FUNCTION_BLOCK FB 120
VERSION : 0.1
VAR_INPUT
  IN_Cm_ON : BOOL ;	//1: Attiva il ciclo; 0: Reset del ciclo
  IN_HOLD : BOOL ;	//Blocca il ciclo nel passo successivo
  IN_STEP : BOOL ;
END_VAR
VAR_OUTPUT
  OUT_St_CicloInCorso : BOOL ;
  OUT_St_CicloTerminatoOK : BOOL ;
  OUT_St_CicloTerminatoKO : BOOL ;
  OUT_CicloStato : INT ;
  OUT_Page : INT ;
  OUT_Message : INT ;
END_VAR
VAR
  Stato : INT ;
  StatoSeguente : INT ;
  FrontePassoSingolo : BOOL ;
  Stat_CicloTermOk : BOOL ;
  Stat_CicloTermKO : BOOL ;
  Stat_CicloInCorso : BOOL ;
  Timer_Pennarello : SFB 4;
END_VAR
VAR_TEMP
  Pag_Active : ARRAY  [0 .. 100 ] OF BOOL ;
END_VAR
BEGIN
NETWORK
TITLE = FLOW CHART
NETWORK
TITLE = Update state
      A     #IN_Cm_ON;
      JC    M002;
      L     0;
      T     #Stato;
      T     #StatoSeguente;
M002: NOP   0;
//->Update State
      A     #IN_STEP;
      FP    #FrontePassoSingolo;
      ON    #IN_HOLD;	//se usassi UN l'Hold agirebbe anche su avanzamento a passo singolo 
      JCN   N100;
      L     #StatoSeguente;
      T     #Stato;
N100: NOP   0;
// determinazione bit di stato
      CALL  FC 17 (
           Valore                   := #Stato,
           States                   := P#DB120.DBX 8.0 BYTE 8);
NETWORK
TITLE = Detect page active from OP
// serve??????
//      CALL  "Conv_INT->BIT"
//       Valore:=DB325.DBW2
//       States:=#Pag_Active
NETWORK
TITLE = States particular
      L     #Stato;
      L     0;
      <>I;
//->Evita ritardi
      A     #IN_Cm_ON;
      =     #Stat_CicloInCorso;
      A     DB120.DBX 15.4;
      =     #Stat_CicloTermOk;
      A     DB120.DBX 37.7;
      =     #Stat_CicloTermKO;
NETWORK
TITLE = Diagnostic default
//    L     0
//    T     #Page
//    L     0
//    T     #Message 
//      L     6
//      T     #StatoSeguente
NETWORK
TITLE = State <0>: Ciclo off
      A     DB120.DBX 8.0;
      A     #IN_Cm_ON;
      JC    A000;
      L     DB120.DBW 2;
      T     #OUT_Page;
      L     1;	// Ciclo off
      T     #OUT_Message;
      JU    Z000;
A000: L     10;
      T     #StatoSeguente;
Z000: NOP   0;
NETWORK
TITLE = State <10>: Inserimento pezzi su attrezzo e start ciclo
      A     DB120.DBX 9.2;
      JCN   Z010;
      A     DB101.DBX 0.6;
      A     DB101.DBX 0.4;
      A     DB106.DBX 0.7;
      A     DB106.DBX 1.0;
      AN    DB106.DBX 1.1;
      A     DB106.DBX 1.2;
      AN    DB106.DBX 1.3;
      A     DB106.DBX 1.4;
      AN    DB106.DBX 1.5;
      A     DB105.DBX 0.6;
      JC    Y010;
// Messaggi
// Inserisci spacer correttamente
      AN    DB106.DBX 1.0;
      ON    DB106.DBX 1.2;
      ON    DB106.DBX 1.4;
      JC    A010;
// almeno uno Spacer inserito male
      A     DB106.DBX 1.1;
      O     DB106.DBX 1.3;
      O     DB106.DBX 1.3;
      JC    B010;
// Inserisci nozzle ring
      AN    DB106.DBX 0.7;
      JC    C010;
// Start ciclo per Bloccare il pezzo
      JU    D010;
A010: L     DB120.DBW 2;
      T     #OUT_Page;
      L     2;	// Inserisci spacer correttamente
      T     #OUT_Message;
      JU    Z010;
B010: L     DB120.DBW 2;
      T     #OUT_Page;
      L     3;	// almeno uno Spacer inserito male
      T     #OUT_Message;
      JU    Z010;
C010: L     DB120.DBW 2;
      T     #OUT_Page;
      L     4;	// Inserisci nozzle ring
      T     #OUT_Message;
      JU    Z010;
D010: L     DB120.DBW 2;
      T     #OUT_Page;
      L     5;	// Start ciclo per Bloccare il pezzo
      T     #OUT_Message;
      JU    Z010;
// Stati di destinazione
Y010: L     13;
      T     #StatoSeguente;
Z010: NOP   0;
NETWORK
TITLE = State <13>: Blocca Pezzo e sblocca index
      A     DB120.DBX 9.5;
      JCN   Z013;
      A     DB101.DBX 0.5;
      A     DB101.DBX 0.3;
      A(;
      A     DB105.DBX 11.3;
      O     DB105.DBX 11.7;
      );
      A     DB105.DBX 10.2;
      JC    Y013;
// Messaggi
// Blocco pezzo e sblocco cassetto in corso
      AN    DB101.DBX 0.5;
      ON    DB101.DBX 0.3;
      JC    A013;
// Porta cassetto in zona di lavorazione
      AN    DB105.DBX 10.2;
      JC    B013;
      JU    B013;
A013: L     DB120.DBW 2;
      T     #OUT_Page;
      L     6;	// Blocco pezzo e sblocco cassetto in corso
      T     #OUT_Message;
      JU    Z013;
B013: L     DB120.DBW 2;
      T     #OUT_Page;
      L     7;	// Porta cassetto in zona di lavorazione
      T     #OUT_Message;
      JU    Z013;
// Stati di destinazione
Y013: L     16;
      T     #StatoSeguente;
Z013: NOP   0;
NETWORK
TITLE = State <16>: Blocca cassetto e prenota ribaditrice
      A     DB120.DBX 10.0;
      JCN   Z016;
      A     DB101.DBX 0.5;
      A     DB101.DBX 0.4;
      A     DB105.DBX 10.2;
      A     DB105.DBX 11.0;
      JC    Y016;
// Messaggi
// Blocco cassetto in corso
      AN    DB101.DBX 0.5;
      ON    DB101.DBX 0.4;
      ON    DB105.DBX 10.2;
      JC    A016;
// Attesa prenotazione ribaditrice
      AN    DB105.DBX 11.0;
      JC    B016;
      JU    B016;
A016: L     DB120.DBW 2;
      T     #OUT_Page;
      L     8;	// Blocco cassetto in corso
      T     #OUT_Message;
      JU    Z016;
B016: L     DB120.DBW 2;
      T     #OUT_Page;
      L     9;	//  Attesa prenotazione ribaditrice
      T     #OUT_Message;
      JU    Z016;
// Stati di destinazione
Y016: L     20;
      T     #StatoSeguente;
Z016: NOP   0;
NETWORK
TITLE = State <20>: Vai a quota di ribaditura punto corrente
      A     DB120.DBX 10.4;
      JCN   Z020;
      A     DB105.DBX 11.1;
      A     DB105.DBX 11.5;
      JC    Y020;
// Messaggi
// Posizionamento assi
      L     DB120.DBW 2;
      T     #OUT_Page;
      L     14;	// Posizionamento assi
      T     #OUT_Message;
      JU    Z020;
// Stati di destinazione
Y020: L     25;
      T     #StatoSeguente;
Z020: NOP   0;
NETWORK
TITLE = State <25>: Esegui ribaditura punto corrente
      A     DB120.DBX 11.1;
      JCN   Z025;
      A     DB105.DBX 11.2;
      JC    Y025;
// Messaggi
// Ribaditura spacer in corso
      L     DB120.DBW 2;
      T     #OUT_Page;
      L     9;	// Ribaditura spacer in corso
      T     #OUT_Message;
      JU    Z025;
// Stati di destinazione
Y025: L     30;
      T     #StatoSeguente;
Z025: NOP   0;
NETWORK
TITLE = State <30>: Risali ribaditrice
      A     DB120.DBX 11.6;
      JCN   Z030;
      A     DB105.DBX 11.3;
      A(;
      L     DB105.DBW 20;
      L     DB110.DBW 80;
      <I;
      );
      JC    Y030;
      A     DB105.DBX 11.3;
      A(;
      L     DB105.DBW 20;
      L     DB110.DBW 80;
      >=I;
      );
      JC    X030;
// Messaggi
// Ribaditura spacer in corso
      L     DB120.DBW 2;
      T     #OUT_Page;
      L     9;	// Ribaditura spacer in corso
      T     #OUT_Message;
      JU    Z030;
// Stati di destinazione
Y030: L     20;
      T     #StatoSeguente;
      JU    Z030;
X030: L     35;
      T     #StatoSeguente;
Z030: NOP   0;
NETWORK
TITLE = State <35>: Sblocco index e cassetto fuori
      A     DB120.DBX 12.3;
      JCN   Z035;
      A     DB101.DBX 0.3;
      A     DB105.DBX 10.3;
      JC    Y035;
// Messaggi
// Sblocco index in corso
      AN    DB101.DBX 0.3;
      JC    A035;
// Porta cassetto in zona di carico
      JU    B035;
A035: L     DB120.DBW 2;
      T     #OUT_Page;
      L     10;	// Sblocco index in corso
      T     #OUT_Message;
      JU    Z035;
B035: L     DB120.DBW 2;
      T     #OUT_Page;
      L     11;	// Porta cassetto in zona di carico
      T     #OUT_Message;
      JU    Z035;
// Stati di destinazione
Y035: L     40;
      T     #StatoSeguente;
Z035: NOP   0;
NETWORK
TITLE = State <40>: Sblocco pezzo e fine lavorazione
      A     DB120.DBX 13.0;
      JCN   Z040;
      A     DB101.DBX 0.4;
      A     DB101.DBX 0.6;
      A     DB105.DBX 10.3;
      AN    DB106.DBX 0.7;
      AN    DB106.DBX 1.0;
      AN    DB106.DBX 1.2;
      AN    DB106.DBX 1.4;
      JC    Y040;
// Messaggi
// Blocco index e sblocco pezzo in corso
      AN    DB101.DBX 0.4;
      ON    DB101.DBX 0.6;
      JC    A040;
// Rimuovi pezzo buono dalla stazione
      JU    B040;
A040: L     DB120.DBW 2;
      T     #OUT_Page;
      L     12;	// Blocco index e sblocco pezzo in corso
      T     #OUT_Message;
      JU    Z040;
B040: L     DB120.DBW 2;
      T     #OUT_Page;
      L     13;	// Rimuovi pezzo buono dalla stazione
      T     #OUT_Message;
      JU    Z040;
// Stati di destinazione
Y040: L     60;
      T     #StatoSeguente;
Z040: NOP   0;
NETWORK
TITLE =
      A     DB120.DBX 15.4;
      JCN   Z060;
// Stati di destinazione
      L     10;
      T     #StatoSeguente;
Z060: NOP   0;
NETWORK
TITLE = Output
      L     #Stato;
      T     #OUT_CicloStato;
      A     #Stat_CicloInCorso;
      =     #OUT_St_CicloInCorso;
      A     #Stat_CicloTermOk;
      =     #OUT_St_CicloTerminatoOK;
      A     #Stat_CicloTermKO;
      =     #OUT_St_CicloTerminatoKO;
END_FUNCTION_BLOCK

FUNCTION_BLOCK FB 121
VERSION : 0.1
VAR_INPUT
  IN_Cm_ON : BOOL ;	//1: Attiva il ciclo; 0: Reset del ciclo
  IN_HOLD : BOOL ;	//Blocca il ciclo nel passo successivo
  IN_STEP : BOOL ;
END_VAR
VAR_OUTPUT
  OUT_St_CicloInCorso : BOOL ;
  OUT_St_CicloTerminatoOK : BOOL ;
  OUT_St_CicloTerminatoKO : BOOL ;
  OUT_CicloStato : INT ;
  OUT_Page : INT ;
  OUT_Message : INT ;
END_VAR
VAR
  Stato : INT ;
  StatoSeguente : INT ;
  FrontePassoSingolo : BOOL ;
  Stat_CicloTermOk : BOOL ;
  Stat_CicloTermKO : BOOL ;
  Stat_CicloInCorso : BOOL ;
  Timer_Pennarello : SFB 4;
END_VAR
VAR_TEMP
  Pag_Active : ARRAY  [0 .. 100 ] OF BOOL ;
END_VAR
BEGIN
NETWORK
TITLE = FLOW CHART
NETWORK
TITLE = Update state
      A     #IN_Cm_ON;
      JC    M002;
      L     0;
      T     #Stato;
      T     #StatoSeguente;
M002: NOP   0;
//->Update State
      A     #IN_STEP;
      FP    #FrontePassoSingolo;
      ON    #IN_HOLD;	//se usassi UN l'Hold agirebbe anche su avanzamento a passo singolo 
      JCN   N100;
      L     #StatoSeguente;
      T     #Stato;
N100: NOP   0;
// determinazione bit di stato
      CALL  FC 17 (
           Valore                   := #Stato,
           States                   := P#DB120.DBX 30.0 BYTE 8);
NETWORK
TITLE = States particular
      L     #Stato;
      L     0;
      <>I;
//->Evita ritardi
      A     #IN_Cm_ON;
      =     #Stat_CicloInCorso;
      A     DB120.DBX 37.4;
      =     #Stat_CicloTermOk;
      A     DB120.DBX 37.7;
      =     #Stat_CicloTermKO;
NETWORK
TITLE = State <0>: Ciclo off
      A     DB120.DBX 30.0;
      A     #IN_Cm_ON;
      JC    A000;
      L     DB120.DBW 24;
      T     #OUT_Page;
      L     20;	// ciclo off
      T     #OUT_Message;
      JU    Z000;
A000: L     10;
      T     #StatoSeguente;
Z000: NOP   0;
NETWORK
TITLE = State <10>: Sali ribaditrice
      A     DB120.DBX 31.2;
      JCN   Z010;
      A     DB105.DBX 11.3;
      O     DB105.DBX 11.7;
      AN    DB101.DBX 0.1;
      JC    Y010;
      A     DB105.DBX 11.3;
      O     DB105.DBX 11.7;
      A     DB101.DBX 0.1;
      JC    X010;
// Messaggi
// Salita ribaditrice in corso
      L     DB120.DBW 24;
      T     #OUT_Page;
      L     21;	// Salita ribaditrice in corso
      T     #OUT_Message;
      JU    Z010;
// Stati di destinazione
Y010: L     15;
      T     #StatoSeguente;
      JU    Z010;
X010: L     20;
      T     #StatoSeguente;
Z010: NOP   0;
NETWORK
TITLE = State <15>: Sblocca index e cassetto fuori
      A     DB120.DBX 31.7;
      JCN   Z015;
      A     DB101.DBX 0.3;
      A     DB105.DBX 10.3;
      JC    Y015;
// Messaggi
//   Sblocco index in corso
      AN    DB101.DBX 0.3;
      JC    A015;
// Porta cassetto in zona di scarico
      JU    B015;
A015: L     DB120.DBW 24;
      T     #OUT_Page;
      L     22;	//  Sblocco index in corso
      T     #OUT_Message;
      JU    Z015;
B015: L     DB120.DBW 24;
      T     #OUT_Page;
      L     23;	// Porta cassetto in zona di scarico
      T     #OUT_Message;
      JU    Z015;
// Stati di destinazione
Y015: L     20;
      T     #StatoSeguente;
Z015: NOP   0;
NETWORK
TITLE = State <20>: Blocca index e sblocca pezzo - rimuovi scarto
      A     DB120.DBX 32.4;
      JCN   Z020;
      A     DB101.DBX 0.6;
      A     DB101.DBX 0.4;
      A     DB105.DBX 10.3;
      AN    DB106.DBX 0.7;
      JC    Y020;
// Messaggi
// Blocco index e sblocco pezzo in corso
      AN    DB101.DBX 0.6;
      ON    DB101.DBX 0.4;
      ON    DB105.DBX 10.3;
      JC    A020;
// Rimuovi pezzo scarto dalla stazione
      JU    B020;
A020: L     DB120.DBW 24;
      T     #OUT_Page;
      L     24;	// Blocco index e sblocco pezzo in corso
      T     #OUT_Message;
      JU    Z020;
B020: L     DB120.DBW 24;
      T     #OUT_Page;
      L     25;	// Rimuovi pezzo scarto dalla stazione
      T     #OUT_Message;
      JU    Z020;
// Stati di destinazione
Y020: L     60;
      T     #StatoSeguente;
Z020: NOP   0;
NETWORK
TITLE = Output
      L     #Stato;
      T     #OUT_CicloStato;
      A     #Stat_CicloInCorso;
      =     #OUT_St_CicloInCorso;
      A     #Stat_CicloTermOk;
      =     #OUT_St_CicloTerminatoOK;
      A     #Stat_CicloTermKO;
      =     #OUT_St_CicloTerminatoKO;
END_FUNCTION_BLOCK

FUNCTION_BLOCK FB 170
VERSION : 0.1
VAR_INPUT
  IN_Cm_ON : BOOL ;	//1: Attiva il ciclo; 0: Reset del ciclo
  IN_HOLD : BOOL ;	//Blocca il ciclo nel passo successivo
  IN_STEP : BOOL ;
END_VAR
VAR_OUTPUT
  OUT_St_CicloInCorso : BOOL ;
  OUT_St_CicloTerminatoOK : BOOL ;
  OUT_St_CicloTerminatoKO : BOOL ;
  OUT_CicloStato : INT ;
  OUT_Page : INT ;
  OUT_Message : INT ;
END_VAR
VAR
  Stato : INT ;
  StatoSeguente : INT ;
  FrontePassoSingolo : BOOL ;
  Stat_CicloTermOk : BOOL ;
  Stat_CicloTermKO : BOOL ;
  Stat_CicloInCorso : BOOL ;
END_VAR
VAR_TEMP
  Pag_Active : ARRAY  [0 .. 100 ] OF BOOL ;
END_VAR
BEGIN
NETWORK
TITLE = FLOW CHART
NETWORK
TITLE = Update state
      A     #IN_Cm_ON;
      JC    M002;
      L     0;
      T     #Stato;
      T     #StatoSeguente;
M002: NOP   0;
//->Update State
      A     #IN_STEP;
      FP    #FrontePassoSingolo;
      ON    #IN_HOLD;	//se usassi UN l'Hold agirebbe anche su avanzamento a passo singolo 
      JCN   N100;
      L     #StatoSeguente;
      T     #Stato;
N100: NOP   0;
// determinazione bit di stato
      CALL  FC 17 (
           Valore                   := #Stato,
           States                   := P#DB170.DBX 8.0 BYTE 8);
NETWORK
TITLE = States particular
      L     #Stato;
      L     0;
      <>I;
//->Evita ritardi
      A     #IN_Cm_ON;
      =     #Stat_CicloInCorso;
      A     DB170.DBX 15.4;
      =     #Stat_CicloTermOk;
      A     DB170.DBX 37.7;
      =     #Stat_CicloTermKO;
NETWORK
TITLE = Diagnostic default
NETWORK
TITLE = State <0>: Ciclo off
      A     DB170.DBX 8.0;
      A     #IN_Cm_ON;
      JC    A000;
      L     DB170.DBW 2;
      T     #OUT_Page;
      L     1;	// Ciclo off
      T     #OUT_Message;
      JU    Z000;
A000: L     10;
      T     #StatoSeguente;
Z000: NOP   0;
NETWORK
TITLE = State <10>: Inserimento pezzi su attrezzo e cassetto dentrro
      A     DB151.DBX 0.2;
      FP    M 52.0;
      =     DB155.DBX 11.7;
      A     DB155.DBX 11.7;
      A     DB170.DBX 9.2;
      S     DB155.DBX 12.0;
      A     DB155.DBX 12.0;
      AN    DB151.DBX 0.2;
      ON    DB170.DBX 9.2;
      R     DB155.DBX 12.0;
      A     DB155.DBX 12.0;
      L     S5T#500MS;
      SD    T 20;
      A     DB170.DBX 9.2;
      JCN   Z010;
      A     T 20;
      JC    Y010;
// Messaggi
// Inserisci pezzi e porta cassetto dentro
      L     DB170.DBW 2;
      T     #OUT_Page;
      L     2;	//  Inserisci pezzi e porta cassetto dentro
      T     #OUT_Message;
      JU    Z010;
// Stati di destinazione
Y010: L     15;
      T     #StatoSeguente;
Z010: NOP   0;
NETWORK
TITLE = State <15>: Blocca cassetto dentrro
      A     DB170.DBX 9.7;
      JCN   Z015;
      A     DB151.DBX 0.2;
      A     DB151.DBX 0.4;
      JC    Y015;
// Messaggi
// Blocco cassetto in corso
      L     DB170.DBW 2;
      T     #OUT_Page;
      L     3;	// Blocco cassetto in corso
      T     #OUT_Message;
      JU    Z015;
// Stati di destinazione
Y015: L     20;
      T     #StatoSeguente;
Z015: NOP   0;
NETWORK
TITLE = State <20>: Discesa gruppo di piantaggio
      A     DB170.DBX 10.4;
      JCN   Z020;
      A     DB151.DBX 0.7;
      JC    Y020;
// Messaggi
// Discesa gruppo di piantaggio
      L     DB170.DBW 2;
      T     #OUT_Page;
      L     4;	// Discesa gruppo di piantaggio
      T     #OUT_Message;
      JU    Z020;
// Stati di destinazione
Y020: L     25;
      T     #StatoSeguente;
Z020: NOP   0;
NETWORK
TITLE = State <25>: Discesa piantaggio
      A     DB170.DBX 11.1;
      JCN   Z025;
      A     DB155.DBX 11.2;
      JC    Y025;
// Messaggi
// Piantaggio in corso
      L     DB170.DBW 2;
      T     #OUT_Page;
      L     5;	// Piantaggio in corso
      T     #OUT_Message;
      JU    Z025;
// Stati di destinazione
Y025: L     30;
      T     #StatoSeguente;
Z025: NOP   0;
NETWORK
TITLE = State <30>: Risalita piantaggio
      A     DB170.DBX 11.6;
      JCN   Z030;
      A     DB151.DBX 1.0;
      A     DB151.DBX 0.6;
      JC    Y030;
// Messaggi
// Risalita pressa in corso
      L     DB170.DBW 2;
      T     #OUT_Page;
      L     6;	// Risalita pressa in corso
      T     #OUT_Message;
      JU    Z030;
// Stati di destinazione
Y030: L     35;
      T     #StatoSeguente;
Z030: NOP   0;
NETWORK
TITLE = State <35>: Sblocco cassetto
      A     DB170.DBX 12.3;
      JCN   Z035;
      A     DB151.DBX 0.3;
      JC    Y035;
// Messaggi
// Sblocco cassetto in corso
      L     DB170.DBW 2;
      T     #OUT_Page;
      L     7;	// Sblocco cassetto in corso
      T     #OUT_Message;
      JU    Z035;
// Stati di destinazione
Y035: L     60;
      T     #StatoSeguente;
Z035: NOP   0;
NETWORK
TITLE =
      A     DB170.DBX 15.4;
      JCN   Z060;
      L     10;
      T     #StatoSeguente;
Z060: NOP   0;
NETWORK
TITLE = Output
      L     #Stato;
      T     #OUT_CicloStato;
      A     #Stat_CicloInCorso;
      =     #OUT_St_CicloInCorso;
      A     #Stat_CicloTermOk;
      =     #OUT_St_CicloTerminatoOK;
      A     #Stat_CicloTermKO;
      =     #OUT_St_CicloTerminatoKO;
END_FUNCTION_BLOCK

FUNCTION_BLOCK FB 171
VERSION : 0.1
VAR_INPUT
  IN_Cm_ON : BOOL ;	//1: Attiva il ciclo; 0: Reset del ciclo
  IN_HOLD : BOOL ;	//Blocca il ciclo nel passo successivo
  IN_STEP : BOOL ;
END_VAR
VAR_OUTPUT
  OUT_St_CicloInCorso : BOOL ;
  OUT_St_CicloTerminatoOK : BOOL ;
  OUT_St_CicloTerminatoKO : BOOL ;
  OUT_CicloStato : INT ;
  OUT_Page : INT ;
  OUT_Message : INT ;
END_VAR
VAR
  Stato : INT ;
  StatoSeguente : INT ;
  FrontePassoSingolo : BOOL ;
  Stat_CicloTermOk : BOOL ;
  Stat_CicloTermKO : BOOL ;
  Stat_CicloInCorso : BOOL ;
END_VAR
VAR_TEMP
  Pag_Active : ARRAY  [0 .. 100 ] OF BOOL ;
END_VAR
BEGIN
NETWORK
TITLE = FLOW CHART
NETWORK
TITLE = Update state
      A     #IN_Cm_ON;
      JC    M002;
      L     0;
      T     #Stato;
      T     #StatoSeguente;
M002: NOP   0;
//->Update State
      A     #IN_STEP;
      FP    #FrontePassoSingolo;
      ON    #IN_HOLD;	//se usassi UN l'Hold agirebbe anche su avanzamento a passo singolo 
      JCN   N100;
      L     #StatoSeguente;
      T     #Stato;
N100: NOP   0;
// determinazione bit di stato
      CALL  FC 17 (
           Valore                   := #Stato,
           States                   := P#DB170.DBX 30.0 BYTE 8);
NETWORK
TITLE = States particular
      L     #Stato;
      L     0;
      <>I;
//->Evita ritardi
      A     #IN_Cm_ON;
      =     #Stat_CicloInCorso;
      A     DB170.DBX 37.4;
      =     #Stat_CicloTermOk;
      A     DB170.DBX 37.7;
      =     #Stat_CicloTermKO;
NETWORK
TITLE = Diagnostic default
NETWORK
TITLE = State <0>: Ciclo off
      A     DB170.DBX 30.0;
      A     #IN_Cm_ON;
      JC    A000;
      L     DB170.DBW 24;
      T     #OUT_Page;
      L     1;	// Ciclo off
      T     #OUT_Message;
      JU    Z000;
A000: L     10;
      T     #StatoSeguente;
Z000: NOP   0;
NETWORK
TITLE = State <10>: Risalita piantaggio
      A     DB170.DBX 31.2;
      JCN   Z010;
      A     DB151.DBX 1.0;
      A     DB151.DBX 0.6;
      JC    Y010;
// Messaggi
// Risalita pressa in corso
      L     DB170.DBW 24;
      T     #OUT_Page;
      L     6;	// Risalita pressa in corso
      T     #OUT_Message;
      JU    Z010;
// Stati di destinazione
Y010: L     15;
      T     #StatoSeguente;
Z010: NOP   0;
NETWORK
TITLE = State <15>: Sblocco cassetto
      A     DB170.DBX 31.7;
      JCN   Z015;
      A     DB151.DBX 0.3;
      JC    Y015;
// Messaggi
// Sblocco cassetto in corso
      L     DB170.DBW 24;
      T     #OUT_Page;
      L     7;	// Sblocco cassetto in corso
      T     #OUT_Message;
      JU    Z015;
// Stati di destinazione
Y015: L     60;
      T     #StatoSeguente;
Z015: NOP   0;
NETWORK
TITLE = Output
      L     #Stato;
      T     #OUT_CicloStato;
      A     #Stat_CicloInCorso;
      =     #OUT_St_CicloInCorso;
      A     #Stat_CicloTermOk;
      =     #OUT_St_CicloTerminatoOK;
      A     #Stat_CicloTermKO;
      =     #OUT_St_CicloTerminatoKO;
END_FUNCTION_BLOCK

FUNCTION_BLOCK FB 220
VERSION : 0.1
VAR_INPUT
  IN_Cm_ON : BOOL ;	//1: Attiva il ciclo; 0: Reset del ciclo
  IN_HOLD : BOOL ;	//Blocca il ciclo nel passo successivo
  IN_STEP : BOOL ;
END_VAR
VAR_OUTPUT
  OUT_St_CicloInCorso : BOOL ;
  OUT_St_CicloTerminatoOK : BOOL ;
  OUT_St_CicloTerminatoKO : BOOL ;
  OUT_CicloStato : INT ;
  OUT_Page : INT ;
  OUT_Message : INT ;
END_VAR
VAR
  Stato : INT ;
  StatoSeguente : INT ;
  FrontePassoSingolo : BOOL ;
  Stat_CicloTermOk : BOOL ;
  Stat_CicloTermKO : BOOL ;
  Stat_CicloInCorso : BOOL ;
  Timer_Pennarello : SFB 4;
END_VAR
VAR_TEMP
  Pag_Active : ARRAY  [0 .. 100 ] OF BOOL ;
END_VAR
BEGIN
NETWORK
TITLE = FLOW CHART
NETWORK
TITLE = Update state
      A     #IN_Cm_ON;
      JC    M002;
      L     0;
      T     #Stato;
      T     #StatoSeguente;
M002: NOP   0;
//->Update State
      A     #IN_STEP;
      FP    #FrontePassoSingolo;
      ON    #IN_HOLD;	//se usassi UN l'Hold agirebbe anche su avanzamento a passo singolo 
      JCN   N100;
      L     #StatoSeguente;
      T     #Stato;
N100: NOP   0;
// determinazione bit di stato
      CALL  FC 17 (
           Valore                   := #Stato,
           States                   := P#DB220.DBX 8.0 BYTE 8);
NETWORK
TITLE = Detect page active from OP
// serve??????
//      CALL  "Conv_INT->BIT"
//       Valore:=DB325.DBW2
//       States:=#Pag_Active
NETWORK
TITLE = States particular
      L     #Stato;
      L     0;
      <>I;
//->Evita ritardi
      A     #IN_Cm_ON;
      =     #Stat_CicloInCorso;
      A     DB220.DBX 15.4;
      =     #Stat_CicloTermOk;
      A     DB220.DBX 15.7;
      =     #Stat_CicloTermKO;
NETWORK
TITLE = Diagnostic default
//    L     0
//    T     #Page
//    L     0
//    T     #Message 
//      L     6
//      T     #StatoSeguente
NETWORK
TITLE = State <0>: Ciclo off
      A     DB220.DBX 8.0;
      A     #IN_Cm_ON;
      JC    A000;
      L     DB120.DBW 24;
      T     #OUT_Page;
      L     1;	// ciclo off
      T     #OUT_Message;
      JU    Z000;
A000: L     10;
      T     #StatoSeguente;
Z000: NOP   0;
NETWORK
TITLE = State <10>: Inserimento pezzi su attrezzo e start ciclo
      A     DB220.DBX 9.2;
      JCN   Z010;
      A     DB201.DBX 0.7;
      A     DB201.DBX 0.5;
      A     DB205.DBX 0.6;
      JC    Y010;
// Messaggi
// Inserisci nozzle ring e Start ciclo
      L     DB220.DBW 2;
      T     #OUT_Page;
      L     4;	// Inserisci nozzle ring e start ciclo
      T     #OUT_Message;
      JU    Z010;
// Stati di destinazione
Y010: L     11;
      T     #StatoSeguente;
Z010: NOP   0;
NETWORK
TITLE = State <11>: Blocca index e controlla presenza pezzo
      A     DB220.DBX 9.3;
      JCN   Z011;
      A     DB201.DBX 0.6;
      A     DB206.DBX 0.7;
      JC    Y011;
      A     DB205.DBX 0.6;
      JC    X011;
// Messaggi
// Inserisci nozzle ring
      AN    DB206.DBX 0.7;
      JC    A011;
      JU    Z011;
A011: L     DB220.DBW 2;
      T     #OUT_Page;
      L     5;	// Inserisci nozzle ring
      T     #OUT_Message;
      JU    Z011;
// Stati di destinazione
X011: L     10;
      T     #StatoSeguente;
      JU    Z011;
Y011: L     13;
      T     #StatoSeguente;
Z011: NOP   0;
NETWORK
TITLE = State <13>: sblocca index
      A     DB220.DBX 9.5;
      JCN   Z013;
      A     DB201.DBX 0.6;
      A     DB201.DBX 0.4;
      A(;
      A     DB205.DBX 11.3;
      O     DB205.DBX 11.7;
      );
      A     DB205.DBX 10.2;
      A     DB201.DBX 0.1;
      JC    Y013;
// Messaggi
// Blocco pezzo e sblocco cassetto in corso
      AN    DB201.DBX 0.6;
      ON    DB201.DBX 0.4;
      JC    A013;
// Porta cassetto in zona di lavorazione
      AN    DB205.DBX 10.2;
      JC    B013;
      JU    C013;
A013: L     DB220.DBW 2;
      T     #OUT_Page;
      L     6;	// Blocco pezzo e sblocco cassetto in corso
      T     #OUT_Message;
      JU    Z013;
B013: L     DB220.DBW 2;
      T     #OUT_Page;
      L     7;	// Porta cassetto in zona di lavorazione
      T     #OUT_Message;
      JU    Z013;
C013: L     DB220.DBW 2;
      T     #OUT_Page;
      L     3;	// Controlla presenza Pipe
      T     #OUT_Message;
      JU    Z013;
// Stati di destinazione
Y013: L     16;
      T     #StatoSeguente;
Z013: NOP   0;
NETWORK
TITLE = State <16>: Blocca cassetto e prenota ribaditrice
      A     DB220.DBX 10.0;
      JCN   Z016;
      A     DB201.DBX 0.6;
      A     DB201.DBX 0.5;
      A     DB205.DBX 10.2;
      A     DB205.DBX 11.0;
      JC    Y016;
// Messaggi
// Blocco cassetto in corso
      AN    DB201.DBX 0.6;
      ON    DB201.DBX 0.5;
      ON    DB205.DBX 10.2;
      JC    A016;
// Attesa prenotazione ribaditrice
      AN    DB205.DBX 11.0;
      JC    B016;
      JU    B016;
A016: L     DB220.DBW 2;
      T     #OUT_Page;
      L     8;	// Blocco cassetto in corso
      T     #OUT_Message;
      JU    Z016;
B016: L     DB220.DBW 2;
      T     #OUT_Page;
      L     9;	//  Attesa prenotazione ribaditrice
      T     #OUT_Message;
      JU    Z016;
// Stati di destinazione
Y016: L     20;
      T     #StatoSeguente;
Z016: NOP   0;
NETWORK
TITLE = State <20>: Vai a quota di ribaditura punto corrente
      A     DB220.DBX 10.4;
      JCN   Z020;
      A     DB205.DBX 11.1;
      A     DB205.DBX 11.5;
      JC    Y020;
// Messaggi
// Posizionamento assi
      L     DB220.DBW 2;
      T     #OUT_Page;
      L     15;	// Posizionamento assi
      T     #OUT_Message;
      JU    Z020;
// Stati di destinazione
Y020: L     25;
      T     #StatoSeguente;
Z020: NOP   0;
NETWORK
TITLE = State <25>: Esegui ribaditura punto corrente
      A     DB220.DBX 11.1;
      JCN   Z025;
      A     DB205.DBX 11.2;
      JC    Y025;
// Messaggi
// Ribaditura spacer in corso
      L     DB220.DBW 2;
      T     #OUT_Page;
      L     10;	// Ribaditura spacer in corso
      T     #OUT_Message;
      JU    Z025;
// Stati di destinazione
Y025: L     30;
      T     #StatoSeguente;
Z025: NOP   0;
NETWORK
TITLE = State <30>: Risali ribaditrice
      A     DB220.DBX 11.6;
      JCN   Z030;
      A     DB205.DBX 11.3;
      A(;
      L     DB205.DBW 20;
      L     DB210.DBW 80;
      <I;
      );
      JC    Y030;
      A     DB205.DBX 11.3;
      A(;
      L     DB205.DBW 20;
      L     DB210.DBW 80;
      >=I;
      );
      JC    X030;
// Messaggi
// Ribaditura spacer in corso
      L     DB220.DBW 2;
      T     #OUT_Page;
      L     10;	// Ribaditura spacer in corso
      T     #OUT_Message;
      JU    Z030;
// Stati di destinazione
Y030: L     20;
      T     #StatoSeguente;
      JU    Z030;
X030: L     35;
      T     #StatoSeguente;
Z030: NOP   0;
NETWORK
TITLE = State <35>: Sblocco index e cassetto fuori
      A     DB220.DBX 12.3;
      JCN   Z035;
      A     DB201.DBX 0.4;
      A     DB205.DBX 10.3;
      JC    Y035;
// Messaggi
// Sblocco index in corso
      AN    DB201.DBX 0.4;
      JC    A035;
// Porta cassetto in zona di carico
      JU    B035;
A035: L     DB220.DBW 2;
      T     #OUT_Page;
      L     11;	// Sblocco index in corso
      T     #OUT_Message;
      JU    Z035;
B035: L     DB220.DBW 2;
      T     #OUT_Page;
      L     12;	// Porta cassetto in zona di carico
      T     #OUT_Message;
      JU    Z035;
// Stati di destinazione
Y035: L     40;
      T     #StatoSeguente;
Z035: NOP   0;
NETWORK
TITLE = State <40>: Sblocco pezzo e fine lavorazione
      A     DB220.DBX 13.0;
      JCN   Z040;
      A     DB201.DBX 0.5;
      A     DB201.DBX 0.7;
      A     DB205.DBX 10.3;
      AN    DB206.DBX 0.7;
      JC    Y040;
// Messaggi
// Blocco index e sblocco pezzo in corso
      AN    DB201.DBX 0.5;
      ON    DB201.DBX 0.7;
      JC    A040;
// Rimuovi pezzo buono dalla stazione
      JU    B040;
A040: L     DB220.DBW 2;
      T     #OUT_Page;
      L     13;	// Blocco index e sblocco pezzo in corso
      T     #OUT_Message;
      JU    Z040;
B040: L     DB220.DBW 2;
      T     #OUT_Page;
      L     14;	// Rimuovi pezzo buono dalla stazione
      T     #OUT_Message;
      JU    Z040;
// Stati di destinazione
Y040: L     60;
      T     #StatoSeguente;
Z040: NOP   0;
NETWORK
TITLE =
      A     DB220.DBX 15.4;
      JCN   Z060;
// Stati di destinazione
      L     10;
      T     #StatoSeguente;
Z060: NOP   0;
NETWORK
TITLE = Output
      L     #Stato;
      T     #OUT_CicloStato;
      A     #Stat_CicloInCorso;
      =     #OUT_St_CicloInCorso;
      A     #Stat_CicloTermOk;
      =     #OUT_St_CicloTerminatoOK;
      A     #Stat_CicloTermKO;
      =     #OUT_St_CicloTerminatoKO;
END_FUNCTION_BLOCK

FUNCTION_BLOCK FB 221
VERSION : 0.1
VAR_INPUT
  IN_Cm_ON : BOOL ;	//1: Attiva il ciclo; 0: Reset del ciclo
  IN_HOLD : BOOL ;	//Blocca il ciclo nel passo successivo
  IN_STEP : BOOL ;
END_VAR
VAR_OUTPUT
  OUT_St_CicloInCorso : BOOL ;
  OUT_St_CicloTerminatoOK : BOOL ;
  OUT_St_CicloTerminatoKO : BOOL ;
  OUT_CicloStato : INT ;
  OUT_Page : INT ;
  OUT_Message : INT ;
END_VAR
VAR
  Stato : INT ;
  StatoSeguente : INT ;
  FrontePassoSingolo : BOOL ;
  Stat_CicloTermOk : BOOL ;
  Stat_CicloTermKO : BOOL ;
  Stat_CicloInCorso : BOOL ;
  Timer_Pennarello : SFB 4;
END_VAR
VAR_TEMP
  Pag_Active : ARRAY  [0 .. 100 ] OF BOOL ;
END_VAR
BEGIN
NETWORK
TITLE = FLOW CHART
NETWORK
TITLE = Update state
      A     #IN_Cm_ON;
      JC    M002;
      L     0;
      T     #Stato;
      T     #StatoSeguente;
M002: NOP   0;
//->Update State
      A     #IN_STEP;
      FP    #FrontePassoSingolo;
      ON    #IN_HOLD;	//se usassi UN l'Hold agirebbe anche su avanzamento a passo singolo 
      JCN   N100;
      L     #StatoSeguente;
      T     #Stato;
N100: NOP   0;
// determinazione bit di stato
      CALL  FC 17 (
           Valore                   := #Stato,
           States                   := P#DB220.DBX 30.0 BYTE 8);
NETWORK
TITLE = Detect page active from OP
// serve??????
//      CALL  "Conv_INT->BIT"
//       Valore:=DB325.DBW2
//       States:=#Pag_Active
NETWORK
TITLE = States particular
      L     #Stato;
      L     0;
      <>I;
//->Evita ritardi
      A     #IN_Cm_ON;
      =     #Stat_CicloInCorso;
      A     DB220.DBX 37.4;
      =     #Stat_CicloTermOk;
      A     DB220.DBX 37.7;
      =     #Stat_CicloTermKO;
NETWORK
TITLE = Diagnostic default
//    L     0
//    T     #Page
//    L     0
//    T     #Message 
//      L     6
//      T     #StatoSeguente
NETWORK
TITLE = State <0>: Ciclo off
      A     DB220.DBX 30.0;
      A     #IN_Cm_ON;
      JC    A000;
      L     DB120.DBW 24;
      T     #OUT_Page;
      L     20;	// ciclo off
      T     #OUT_Message;
      JU    Z000;
A000: L     10;
      T     #StatoSeguente;
Z000: NOP   0;
NETWORK
TITLE = State <10>: Sali ribaditrice
      A     DB220.DBX 31.2;
      JCN   Z010;
      A     DB205.DBX 11.3;
      O     DB205.DBX 11.7;
      AN    DB201.DBX 0.2;
      JC    Y010;
      A     DB205.DBX 11.3;
      O     DB205.DBX 11.7;
      A     DB201.DBX 0.2;
      JC    X010;
// Messaggi
// Salita ribaditrice in corso
//      UN    "Op40.Bench.Systems".State.Ribaditrice_alta
//      UN    DB205.DBX    11.7
//      SPA   A010
      L     DB220.DBW 24;
      T     #OUT_Page;
      L     21;	// Salita ribaditrice in corso
      T     #OUT_Message;
      JU    Z010;
// Stati di destinazione
Y010: L     15;
      T     #StatoSeguente;
      JU    Z010;
X010: L     20;
      T     #StatoSeguente;
Z010: NOP   0;
NETWORK
TITLE = State <15>: Sblocca index e cassetto fuori
      A     DB220.DBX 31.7;
      JCN   Z015;
      A     DB201.DBX 0.4;
      A     DB205.DBX 10.3;
      JC    Y015;
// Messaggi
//   Sblocco index in corso
      AN    DB201.DBX 0.4;
      JC    A015;
// Porta cassetto in zona di scarico
      JU    B015;
A015: L     DB220.DBW 24;
      T     #OUT_Page;
      L     22;	//  Sblocco index in corso
      T     #OUT_Message;
      JU    Z015;
B015: L     DB220.DBW 24;
      T     #OUT_Page;
      L     23;	// Porta cassetto in zona di scarico
      T     #OUT_Message;
      JU    Z015;
// Stati di destinazione
Y015: L     20;
      T     #StatoSeguente;
Z015: NOP   0;
NETWORK
TITLE = State <20>: Blocca index e sblocca pezzo - rimuovi scarto
      A     DB220.DBX 32.4;
      JCN   Z020;
      A     DB201.DBX 0.7;
      A     DB201.DBX 0.5;
      A     DB205.DBX 10.3;
      AN    DB206.DBX 0.7;
      JC    Y020;
// Messaggi
// Blocco index e sblocco pezzo in corso
      AN    DB201.DBX 0.7;
      ON    DB201.DBX 0.5;
      ON    DB205.DBX 10.3;
      JC    A020;
// Rimuovi pezzo scarto dalla stazione
      JU    B020;
A020: L     DB220.DBW 24;
      T     #OUT_Page;
      L     24;	// Blocco index e sblocco pezzo in corso
      T     #OUT_Message;
      JU    Z020;
B020: L     DB220.DBW 24;
      T     #OUT_Page;
      L     25;	// Rimuovi pezzo scarto dalla stazione
      T     #OUT_Message;
      JU    Z020;
// Stati di destinazione
Y020: L     60;
      T     #StatoSeguente;
Z020: NOP   0;
NETWORK
TITLE = Output
      L     #Stato;
      T     #OUT_CicloStato;
      A     #Stat_CicloInCorso;
      =     #OUT_St_CicloInCorso;
      A     #Stat_CicloTermOk;
      =     #OUT_St_CicloTerminatoOK;
      A     #Stat_CicloTermKO;
      =     #OUT_St_CicloTerminatoKO;
END_FUNCTION_BLOCK

FUNCTION_BLOCK FB 450
//Gestione di sistema di max 4 assi (X-Y-Z-U) mediante SIEMENS SINAMICS CU320 
//
AUTHOR : Castel
VERSION : 0.1
VAR_INPUT
  Enable_Function : BOOL ;	//Abilitazione esecuzione blocco
  AddrIN : WORD ;
  AddrOUT : WORD ;
  Cmd_Jog_Minus_Axis : BOOL ;	//Start movimento incrementale negativa asse
  Cmd_Jog_Plus_Axis : BOOL ;	//Start movimento incrementale positiva asse
  Cmd_Start_Posit_Axis : BOOL ;	//Muovi alla posizione programmata asse
  Cmd_Reference_Axis : BOOL ;	//Ricerca punto di riferimento
  In_Reference_Cam : BOOL ;	//Camma punto di riferimento
  Cmd_Enable_Axis : BOOL ;	//Abbilita la regolazione rampa
  Cmd_ResetAlarm : BOOL ;	//Reset Allarmi
  Cmd_Override_Axis : INT ;	//Valore override 0..100% asse
  Cmd_Acceleration_Axis : INT ;	//Valore accellerazione 0..100% asse
  Cmd_Deceleration_Axis : INT ;	//Valore decellerazione 0..100% asse
  Cmd_Speed_Axis : DINT ;	//Valore velocita asse
  Cmd_Position_Axis : DINT ;	//Posizione assoluta da raggiungere in micron asse
  Cmd_Positioning_Mode : INT ;	//0=Assoluto, 1=relativo, 2=AssolutoPiu, 3 AssolutoMeno
END_VAR
VAR_OUTPUT
  Profibus_Write_Error : BOOL ;	//Errore nella scrittura dati nella rete Profibus
  Profibus_Read_Error : BOOL ;	//Errore nella lettura dati dalla rete Profibus
  St_Referenced_Axis : BOOL ;	//Arre referenziato
  St_Pos_Axis_OK : BOOL ;	//Posizione asse raggiunta
  St_Axis_Running : BOOL ;	//Asse in movimento
  St_Alarm_Code_Axis : BYTE ;	//Rispote d'errore in codice dall'asse
  St_Position_Axis : DINT ;	//Posizione assoluta asse in micron
  St_EndstrokePlus_Reached : BOOL ;
  St_EndstrokeMinu_Reached : BOOL ;
  St_Axis_ReadyToStart : BOOL ;
END_VAR
VAR
  Asse_ERR_Ricezione : BOOL ;
  Asse_ERR_Trasmissione : BOOL ;
  AsseMossoInPosizioname : BOOL ;
  Axis_Buffer : UDT 450;
END_VAR
VAR_TEMP
  RET_VAL_Write_Axis : INT ;	//Valore di ritorno per diagnosi SFC
  RET_VAL_Read_Axis : INT ;	//Valore di ritorno per diagnosi SFC
  Override_Axis : INT ;
  Acceleration_Axis : INT ;
  Deceleration_Axis : INT ;
  Speed_Axis : DINT ;
END_VAR
BEGIN
NETWORK
TITLE =
      A     #Enable_Function;
      JCN   m000;
NETWORK
TITLE = Lettura dati SINAMICS ASSE X
//Utilizzato Telegramma SIEMENS 110, PZD-12/7
      BLD   7;
      =     L 18.0;	// Byte 310       // Indirizzo iniziale di lettura dalla config. Hw convertito in Hex.
      TAR2  LD 14;
      L     #AddrIN;	//#P_Buffer               //P#DB141.DBX0.0 BYTE 14
      T     LW 19;
      L     W#16#1002;
      T     LW 21;
      L     14;
      T     LW 23;
      L     DINO;
      T     LW 25;
      +AR2  P#34.0;
      TAR2;
      LAR2  LD 14;
      T     LD 27;
      UC    SFC 14;
      {     P#L 19.0, P#L 2.0, P#L 21.0 };
      LAR2  LD 14;
      BLD   8;
NETWORK
TITLE = Anomalia ricezione dati SINAMICS ASSE X
      A(;
      L     #RET_VAL_Read_Axis;
      L     W#16#8000;
      >=I;
      );
      A(;
      L     #RET_VAL_Read_Axis;
      L     W#16#8FFF;
      <=I;
      );
      =     #Asse_ERR_Ricezione;
NETWORK
TITLE =
//***************************** ASSE X **************************************
NETWORK
TITLE = Override asse X
//Campo di lavoro del parametro accellerazione 0..100%
      L     #Cmd_Override_Axis;
      T     #Override_Axis;
      L     #Override_Axis;
      L     100;
      >I;
      JCN   m010;
      L     100;
      T     #Override_Axis;
m010: NOP   0;
      L     #Override_Axis;
      L     0;
      <I;
      JCN   m011;
      L     0;
      T     #Override_Axis;
m011: NOP   0;
      L     #Override_Axis;	// VALORE 0-100% OVERRIDE VALORE DI COMANDO
      ITD;
      L     L#32767;
      *D;
      L     L#100;
      /D;
      T     DIW [AR2,P#56.0];	//  "Telegramma Asse X".OUT.OUT_PZD5    // override max  0..32767    
NETWORK
TITLE = MDI Accelerazione asse X
//Campo di lavoro del parametro accellerazione 0..100%
      L     #Cmd_Acceleration_Axis;
      T     #Acceleration_Axis;
      L     #Acceleration_Axis;
      L     100;
      >I;
      JCN   m020;
      L     100;
      T     #Acceleration_Axis;
m020: NOP   0;
      L     #Acceleration_Axis;
      L     0;
      <I;
      JCN   m021;
      L     0;
      T     #Acceleration_Axis;
m021: NOP   0;
      L     #Acceleration_Axis;	//VALORE 0-100% ACCELERAZIONE VALORE DI COMANDO
      ITD;
      L     L#32767;
      *D;
      L     L#100;
      /D;
      T     DIW [AR2,P#66.0];	//  "Telegramma Asse X".OUT.OUT_PZD10    // MDI accelerazione max  0..32767  
NETWORK
TITLE = MDI Decelerazione asse X
//Campo di lavoro del parametro accellerazione 0..100%
      L     #Cmd_Deceleration_Axis;
      T     #Deceleration_Axis;
      L     #Deceleration_Axis;
      L     100;
      >I;
      JCN   m030;
      L     100;
      T     #Deceleration_Axis;
m030: NOP   0;
      L     #Deceleration_Axis;
      L     0;
      <I;
      JCN   m031;
      L     0;
      T     #Deceleration_Axis;
m031: NOP   0;
      L     #Deceleration_Axis;	//VALORE 0-100% DECELERAZIONE VALORE DI COMANDO
      ITD;
      L     L#32767;
      *D;
      L     L#100;
      /D;
      T     DIW [AR2,P#68.0];	// "Telegramma Asse X".OUT.OUT_PZD11    // MDI decelerazione max  0..32767  
NETWORK
TITLE = MDI Velocità asse X
//Campo di lavoro del parametro decellerazione 0..100%
      L     #Cmd_Speed_Axis;
      T     #Speed_Axis;
      L     #Speed_Axis;
      L     L#30000;
      >D;
      JCN   m040;
      L     L#30000;
      T     #Speed_Axis;
m040: NOP   0;
      L     #Speed_Axis;
      L     L#0;
      <D;
      JCN   m041;
      L     L#0;
      T     #Speed_Axis;
m041: NOP   0;
      L     #Speed_Axis;	//VALORE 0-100% VELOCITA' VALORE DI COMANDO
      T     DID [AR2,P#62.0];	// "Telegramma Asse X".OUT.OUT_PZD8_9    // MDI velocità max  0..30000 
NETWORK
TITLE = MDI Posizione da raggiungere asse X
      L     #Cmd_Position_Axis;
      T     DID [AR2,P#58.0];	// "Telegramma Asse X".OUT.OUT_PZD6_7    // Posizione assoluta da raggiungere un micron
NETWORK
TITLE = MDI Mode asse (Assoluto o Relativo)
//xx0x hex -> assoluto
//xx1x hex -> relativo
//xx2x hex -> ass_pos (solo per correzione modulo)
//xx3x hex -> ass_neg (solo per correzione modulo)
//
// Default posizionamento assoluto!!!
      L     #Cmd_Positioning_Mode;
      JL    Mox;
      JU    Mo0;
      JU    Mo1;
      JU    Mo2;
      JU    Mo3;
Mox:  JU    Mo0;
Mo0:  L     0;	// Posizionamento assoluto
      JU    MoR;
Mo1:  L     W#16#10;	// Posizionamento relativo
      JU    MoR;
Mo2:  L     W#16#20;	// Posizionamento assoluto Più (con modulo)
      JU    MoR;
Mo3:  L     W#16#30;	// Posizionamento assoluto Meno (con modulo)
      JU    MoR;
MoR:  T     DIW [AR2,P#70.0];
NETWORK
TITLE = PACO1 gestione parola di comando 1 asse X
//
//
//
//
// PACO1 Bit10 controllo da plc (abilitazione profibus)
      SET;
      =     DIX [AR2,P#48.2];	// conduzione profibus    
      =     DIX [AR2,P#49.5];	// NO Arresto immediato
      =     DIX [AR2,P#50.7];	// abilita rampa 
// Reset alarm
      A     #Cmd_ResetAlarm;
      =     DIX [AR2,P#49.7];	// "Telegramma Asse X".OUT.OUT_PZD1_BIT7
// Abilitazione asse
      A     #Cmd_Enable_Axis;
      =     DIX [AR2,P#49.1];
      =     DIX [AR2,P#49.2];
      =     DIX [AR2,P#49.3];	// "Telegramma Asse X".OUT.OUT_PZD1_BIT3    // Abilita al funzionamento 
      A     #Cmd_Enable_Axis;
      A     DIX [AR2,P#35.4];
      A     DIX [AR2,P#35.5];
      A     DIX [AR2,P#35.0];
      S     DIX [AR2,P#49.0];
      AN    #Cmd_Enable_Axis;
      R     DIX [AR2,P#49.0];
// Marcia a impulsi jog negativo asse
      A     #Cmd_Jog_Minus_Axis;
      AN    #Cmd_Jog_Plus_Axis;
      AN    #Cmd_Reference_Axis;
      AN    #Cmd_Start_Posit_Axis;
      =     DIX [AR2,P#48.0];	// jog negativo        
// Marcia a impulsi jog positivo asse
      AN    #Cmd_Jog_Minus_Axis;
      A     #Cmd_Jog_Plus_Axis;
      AN    #Cmd_Reference_Axis;
      AN    #Cmd_Start_Posit_Axis;
      =     DIX [AR2,P#48.1];	// jog positivo     
// Ricerca punto di zero
      A     #Cmd_Reference_Axis;
      AN    #Cmd_Jog_Minus_Axis;
      AN    #Cmd_Jog_Plus_Axis;
      AN    #Cmd_Start_Posit_Axis;
      =     DIX [AR2,P#48.3];	// avvio del punto di riferimento  (ricerca zero)
// Camma punto di zero
      A     #In_Reference_Cam;
      =     DIX [AR2,P#53.2];	// Camma di zero
// Comando di marcia
      A     DIX [AR2,P#49.0];	// OFF-1 
      A     DIX [AR2,P#49.1];	// OFF-2
      A     DIX [AR2,P#49.2];	// OFF-3   
      A     DIX [AR2,P#35.0];
      A     DIX [AR2,P#35.1];
      A     DIX [AR2,P#35.2];
      AN    DIX [AR2,P#35.3];
      A     DIX [AR2,P#35.4];
      A     DIX [AR2,P#35.5];
      AN    DIX [AR2,P#35.6];
      AN    #Cmd_Reference_Axis;
      AN    #Cmd_Jog_Minus_Axis;
      AN    #Cmd_Jog_Plus_Axis;
      A     #Cmd_Start_Posit_Axis;
      =     DIX [AR2,P#49.6];	// Attiva movimento
      =     DIX [AR2,P#49.4];	// Rifiuto job di movimento
NETWORK
TITLE = Posizione reale assoluta dell'asse X
      L     DID [AR2,P#44.0];	// "Telegramma Asse X".IN.IN_PZD6_7
      T     #St_Position_Axis;
NETWORK
TITLE = Posizione richiesta raggiunta asse X
// Registra movimento avvenuto asse in posizioamento
      AN    DIX [AR2,P#34.2];
      ON    DIX [AR2,P#34.5];
      A     #Cmd_Start_Posit_Axis;
      S     #AsseMossoInPosizioname;
      AN    #Cmd_Start_Posit_Axis;
      R     #AsseMossoInPosizioname;
      L     #Cmd_Positioning_Mode;
      L     1;
      ==I;
      JC    NABS;
// Controlo posizione raggiunta se posizionamento assoluto
      A(;
      L     DID [AR2,P#44.0];	// "Telegramma Asse X".IN.IN_PZD6_7
      L     L#200;
      +D;
      L     DID [AR2,P#58.0];	// "Telegramma Asse X".OUT.OUT_PZD6_7
      >=D;
      );
      A(;
      L     DID [AR2,P#44.0];	// "Telegramma Asse X".IN.IN_PZD6_7
      L     L#200;
      -D;
      L     DID [AR2,P#58.0];	// "Telegramma Asse X".OUT.OUT_PZD6_7
      <=D;
      );
      A     DIX [AR2,P#34.2];
      A     DIX [AR2,P#34.5];
      A     #Cmd_Start_Posit_Axis;
      =     #St_Pos_Axis_OK;
      JU    FPOK;
NABS: NOP   0;
// Controlo posizione raggiunta se posizionamento relativo
      A     DIX [AR2,P#34.2];
      A     DIX [AR2,P#34.5];
      A     #Cmd_Start_Posit_Axis;
      A     #AsseMossoInPosizioname;
      =     #St_Pos_Axis_OK;
FPOK: NOP   0;
NETWORK
TITLE = Asse X in movimento dopo lo start al Job
      A     DIX [AR2,P#39.4];
      O     DIX [AR2,P#39.5];
      =     #St_Axis_Running;
NETWORK
TITLE = Asse referenziato
      A     DIX [AR2,P#34.3];
      =     #St_Referenced_Axis;
NETWORK
TITLE = Segnalazioni errori o anomalie asse X
      A     DIX [AR2,P#35.3];	//  "Telegramma Asse X".IN.IN_PZD1_BIT3
      JC    m063;
      AN    DIX [AR2,P#35.0];	// "Telegramma Asse X".IN.IN_PZD1_BIT0
      JC    m060;
      AN    DIX [AR2,P#35.1];	// "Telegramma Asse X".IN.IN_PZD1_BIT1
      JC    m061;
      AN    DIX [AR2,P#35.2];	// "Telegramma Asse X".IN.IN_PZD1_BIT2
      JC    m062;
      AN    DIX [AR2,P#35.4];	// "Telegramma Asse X".IN.IN_PZD1_BIT4
      JC    m064;
      AN    DIX [AR2,P#35.5];	// "Telegramma Asse X".IN.IN_PZD1_BIT5
      JC    m065;
      A     DIX [AR2,P#35.6];	// "Telegramma Asse X".IN.IN_PZD1_BIT6
      JC    m066;
      A     DIX [AR2,P#39.6];	// "Telegramma Asse X".IN.IN_PZD3_BIT6
      JC    m067;
      A     DIX [AR2,P#39.7];	// "Telegramma Asse X".IN.IN_PZD3_BIT7
      JC    m068;
      JU    m070;
m060: L     1;	// Cod.1: asse non pronto all'inserzione
      JU    m079;
m061: L     2;	// Cod.2: asse non pronto al funzionamento
      JU    m079;
m062: L     3;	// Cod.3: asse non abilitato
      JU    m079;
m063: L     4;	// Cod.4: asse in anomalia
      JU    m079;
m064: L     5;	// Cod.5: asse in arresto per inerzia  (OFF-2)
      JU    m079;
m065: L     6;	// Cod.6: asse in arresto rapido (OFF-3)
      JU    m079;
m066: L     7;	// Cod.7: blocco all'inserzione dell'asse
      JU    m079;
m067: L     8;	// Cod.8: finecorsa SW- raggiunto
      JU    m079;
m068: L     9;	// Cod.9: finecorsa SW+ raggiunto
      JU    m079;
m070: L     0;	// Nessun errore dall'asse
      JU    m079;
m079: T     #St_Alarm_Code_Axis;
NETWORK
TITLE = Invio dati SINAMICS ASSE X
//Utilizzato Telegramma SIEMENS 110, PZD-12/7
      BLD   7;
      =     L 18.0;	//Byte 352       // Indirizzo iniziale di scrittura dalla config. Hw convertito in Hex.
      TAR2  LD 14;
      L     #AddrOUT;
      T     LW 19;
      L     W#16#1002;
      T     LW 21;
      L     24;
      T     LW 23;
      L     DINO;
      T     LW 25;
      +AR2  P#48.0;
      TAR2;
      LAR2  LD 14;
      T     LD 27;
      UC    SFC 15;
      {     P#L 19.0, P#L 21.0, P#L 0.0 };
      LAR2  LD 14;
      BLD   8;
NETWORK
TITLE = Anomalia invio dati SINAMICS ASSE X
      A(;
      L     #RET_VAL_Write_Axis;
      L     W#16#8000;
      >=I;
      );
      A(;
      L     #RET_VAL_Write_Axis;
      L     W#16#8FFF;
      <=I;
      );
      =     #Asse_ERR_Trasmissione;
      NOP   0;
NETWORK
TITLE = Segnalazioni errore profibus
      A     #Asse_ERR_Trasmissione;
      =     #Profibus_Write_Error;
      A     #Asse_ERR_Ricezione;
      =     #Profibus_Read_Error;
NETWORK
TITLE =
      A     DIX [AR2,P#39.7];
      =     #St_EndstrokePlus_Reached;
      A     DIX [AR2,P#39.6];
      =     #St_EndstrokeMinu_Reached;
      A     DIX [AR2,P#35.0];
      A     DIX [AR2,P#35.1];
      A     DIX [AR2,P#35.2];
      A     DIX [AR2,P#34.0];
      A     DIX [AR2,P#34.3];
      =     #St_Axis_ReadyToStart;
NETWORK
TITLE =
m000: NOP   0;
END_FUNCTION_BLOCK

FUNCTION_BLOCK FB 455
//Gestione di sistema assi mediante SIEMENS SINAMICS CU320 
//
VERSION : 0.1
VAR_INPUT
  IN_Enable : BOOL ;	//Abilitazione esecuzione blocco
  IN_Addr_Read : WORD ;	//Indirizzo iniziale di lettura dati da profibus in cod. esadecimale
  IN_Addr_Write : WORD ;	//Indirizzo iniziale di scrittura dati nel profibus in cod. esadecimale
END_VAR
VAR_OUTPUT
  OUT_HW_DI0 : BOOL ;
  OUT_HW_DI1 : BOOL ;
  OUT_HW_DI2 : BOOL ;
  OUT_HW_DI3 : BOOL ;
  OUT_HW_DI4 : BOOL ;
  OUT_HW_DI5 : BOOL ;
  OUT_HW_DI6 : BOOL ;
  OUT_HW_DI7 : BOOL ;
  OUT_HW_DI8 : BOOL ;
  OUT_HW_DI9 : BOOL ;
  OUT_HW_DI10 : BOOL ;
  OUT_HW_DI11 : BOOL ;
  OUT_HW_DI12 : BOOL ;
  OUT_HW_DI13 : BOOL ;
  OUT_HW_DI14 : BOOL ;
  OUT_HW_DI15 : BOOL ;
  OUT_Profibus_Write_Error : BOOL ;	//Errore nella scrittura dati nella rete Profibus
  OUT_Profibus_Read_Error : BOOL ;	//Errore nella lettura dati dalla rete Profibus
END_VAR
VAR
  CU320_ERR_Ricezione : BOOL ;
  CU320_ERR_Trasmissione : BOOL ;
  Cu320_Buffer : UDT 455;
END_VAR
VAR_TEMP
  Dummy : BOOL ;
  RET_VAL_Write_CU320 : INT ;	//Valore di ritorno per diagnosi SFC
  RET_VAL_Read_CU320 : INT ;	//Valore di ritorno per diagnosi SFC
END_VAR
BEGIN
NETWORK
TITLE =
      AN    #IN_Enable;
      R     #OUT_Profibus_Write_Error;
      R     #OUT_Profibus_Read_Error;
      JC    m000;
NETWORK
TITLE = Lettura dati SINAMICS Control unit CU320
//Utilizzato Telegramma SIEMENS 390, PZD-2/2
      BLD   7;
      =     L 10.0;
      TAR2  LD 6;
      L     #IN_Addr_Read;
      T     LW 11;
      L     W#16#1002;
      T     LW 13;
      L     4;
      T     LW 15;
      L     DINO;
      T     LW 17;
      +AR2  P#12.0;
      TAR2;
      LAR2  LD 6;
      T     LD 19;
      UC    SFC 14;
      {     P#L 11.0, P#L 4.0, P#L 13.0 };
      LAR2  LD 6;
      BLD   8;
NETWORK
TITLE = Anomalia ricezione dati SINAMICS Cu320
      A(;
      L     #RET_VAL_Read_CU320;
      L     W#16#8000;
      >=I;
      );
      A(;
      L     #RET_VAL_Read_CU320;
      L     W#16#8FFF;
      <=I;
      );
      =     #CU320_ERR_Ricezione;
NETWORK
TITLE = Parole di stato telegramma Cu320
// Segnale di richiesta reset Sinamics dall'esterno
      A     DIX [AR2,P#15.0];
      =     #OUT_HW_DI8;
      A     DIX [AR2,P#15.1];
      =     #OUT_HW_DI9;
      A     DIX [AR2,P#15.2];
      =     #OUT_HW_DI10;
      A     DIX [AR2,P#15.3];
      =     #OUT_HW_DI11;
      A     DIX [AR2,P#15.4];
      =     #OUT_HW_DI12;
      A     DIX [AR2,P#15.5];
      =     #OUT_HW_DI13;
      A     DIX [AR2,P#15.6];
      =     #OUT_HW_DI14;
      A     DIX [AR2,P#15.7];
      =     #OUT_HW_DI15;
      A     DIX [AR2,P#14.0];
      =     #OUT_HW_DI0;
      A     DIX [AR2,P#14.1];
      =     #OUT_HW_DI1;
      A     DIX [AR2,P#14.2];
      =     #OUT_HW_DI2;
      A     DIX [AR2,P#14.3];
      =     #OUT_HW_DI3;
      A     DIX [AR2,P#14.4];
      =     #OUT_HW_DI4;
      A     DIX [AR2,P#14.5];
      =     #OUT_HW_DI5;
      A     DIX [AR2,P#14.6];
      =     #OUT_HW_DI6;
      A     DIX [AR2,P#14.7];
      =     #OUT_HW_DI7;
NETWORK
TITLE = Segnalazioni errore profibus
//      U     #CU320_ERR_Trasmissione
//      =     #OUT_Profibus_Write_Error
      A     #CU320_ERR_Ricezione;
      =     #OUT_Profibus_Read_Error;
      JU    m001;
m000: CLR;
      =     #OUT_HW_DI0;
      =     #OUT_HW_DI1;
      =     #OUT_HW_DI2;
      =     #OUT_HW_DI3;
      =     #OUT_HW_DI7;
      =     #OUT_HW_DI6;
      =     #OUT_HW_DI5;
      =     #OUT_HW_DI4;
      =     #OUT_HW_DI13;
      =     #OUT_HW_DI14;
      =     #OUT_HW_DI15;
      =     #OUT_HW_DI14;
m001: NOP   0;
NETWORK
TITLE = Azzera uscite con blocco disabilitato
END_FUNCTION_BLOCK

// FC 5: know-how protected block, not included

FUNCTION FC 17 : VOID
AUTHOR : Filip1
NAME : StateBit
VERSION : 1.0
VAR_INPUT
  Valore : INT ;
END_VAR
VAR_IN_OUT
  States : ANY ;
END_VAR
VAR_TEMP
  CONTATORE : WORD ;
  Num_DB : INT ;
  Punt : DWORD ;
  Num_Bit : WORD ;
  Data_T : BYTE ;
  Punt_1 : DWORD ;
END_VAR
BEGIN
NETWORK
TITLE = Decodifica INT -> serie di bit
      L     P##States;
      LAR1;
      L     B [AR1,P#1.0];
      T     #Data_T;
      L     W [AR1,P#2.0];
      T     #Num_Bit;
      L     W [AR1,P#4.0];
      T     #Num_DB;
      L     D [AR1,P#6.0];
      T     #Punt;
      L     #Data_T;
      L     1;	//tipo di dati = 1 -> bool
      ==I;
      JC    OK;
      L     #Data_T;
      L     3;	//tipo di dati = 2 o 3 -> byte o char
      >I;
      JC    no_b;
      L     #Num_Bit;
      L     8;
      *I;
      T     #Num_Bit;
      JC    OK;
no_b: L     #Data_T;
      L     5;	//tipo di dati = 4 o 5 -> int o word
      >I;
      JC    Exit;
      L     #Num_Bit;
      L     16;
      *I;
      T     #Num_Bit;
      JC    OK;
      JCN   Exit;
OK:   OPN   DB [#Num_DB];
      L     #Punt;
      T     #Punt_1;
//- AZZERAMENTO INIZIALE
      L     #Num_Bit;
ZERO: T     #CONTATORE;
      L     #Punt_1;
      LAR1;
      SET;
      R      [AR1,P#0.0];
      L     #Punt_1;
      L     1;
      +D;
      T     #Punt_1;
      L     #CONTATORE;
      LOOP  ZERO;
//- LETTURA BIT DA SETTARE
      L     #Valore;
      L     #Num_Bit;
      <I;
      JCN   Exit;
      L     #Valore;
      L     #Punt;
      +D;
      LAR1;
      SET;
      S      [AR1,P#0.0];
Exit: NOP   0;
END_FUNCTION

FUNCTION FC 20 : VOID
VERSION : 0.1
VAR_INPUT
  Enable : BOOL ;	//Abilita le uscite: sempre a True
  AllarmeEmergenza : BOOL ;	//Presenza allarme di emergenza: se false -> Uscita PlcOk a 0
  AusiliariOK : BOOL ;	//Segnale Ausiliari pronto: per passaggio da modo Emergenza a modo Test Macchina
  ComandoTestMacchina : BOOL ;	//Segnale che forza il modo test Macchina (es. Pulsante di test lampade)
  ComandoSetup : BOOL ;	//Segnale che forza il modo Setuo (es. Selettore di setup)
  ComandoManuale : BOOL ;	//Interruttore con cui si desidera selezionare la modalità manuale
  ComandoAutomatico : BOOL ;	//Interruttore con cui si desidera selezionare la modalità automatica
  TimerTest : TIMER ;	//Timer per test dopo inserzione ausiliari
END_VAR
VAR_OUTPUT
  ModoEmergenza : BOOL ;
  ModoTestMacchina : BOOL ;
  ModoSetup : BOOL ;
  ModoManuale : BOOL ;
  ModoAutomatico : BOOL ;
  DO_PlcOk : BOOL ;
END_VAR
BEGIN
NETWORK
TITLE = Gestioni Modi
NETWORK
TITLE = MacchinaSpenta
      A     #Enable;
      JC    Enbl;
      R     #ModoEmergenza;
      R     #ModoTestMacchina;
      R     #ModoSetup;
      R     #ModoManuale;
      R     #ModoAutomatico;
      R     #DO_PlcOk;
      BEU;
Enbl: NOP   0;
NETWORK
TITLE = CASE Command
      A     #AusiliariOK;
      AN    #AllarmeEmergenza;
      L     S5T#2S;
      SD    #TimerTest;
      AN    #AusiliariOK;
      O     #AllarmeEmergenza;
      JC    Emer;
      A     #AusiliariOK;
      AN    #TimerTest;
      JC    Test;
      A     #TimerTest;
      A     #ComandoSetup;
      JC    Setu;
      A     #TimerTest;
      A(;
      A     #ComandoManuale;
      O     #ModoManuale;
      );
      AN    #ComandoAutomatico;
      JC    Manu;
      A     #TimerTest;
      A(;
      A     #ComandoAutomatico;
      O     #ModoAutomatico;
      );
      AN    #ComandoManuale;
      JC    Auto;
      JU    Setu;
NETWORK
TITLE = CASE: Emergenza
Emer: NOP   0;
      S     #ModoEmergenza;
      R     #ModoTestMacchina;
      R     #ModoSetup;
      R     #ModoManuale;
      R     #ModoAutomatico;
      JU    END;
NETWORK
TITLE = CASE: Test Ausiliari
Test: NOP   0;
      R     #ModoEmergenza;
      S     #ModoTestMacchina;
      R     #ModoSetup;
      R     #ModoManuale;
      R     #ModoAutomatico;
      JU    END;
NETWORK
TITLE = CASE: Modo setup
Setu: NOP   0;
      R     #ModoEmergenza;
      R     #ModoTestMacchina;
      S     #ModoSetup;
      R     #ModoManuale;
      R     #ModoAutomatico;
      JU    END;
NETWORK
TITLE = CASE: Modo Manuale
Manu: NOP   0;
      R     #ModoEmergenza;
      R     #ModoTestMacchina;
      R     #ModoSetup;
      S     #ModoManuale;
      R     #ModoAutomatico;
      JU    END;
NETWORK
TITLE = CASE: Modo Automatico
Auto: NOP   0;
      R     #ModoEmergenza;
      R     #ModoTestMacchina;
      R     #ModoSetup;
      R     #ModoManuale;
      S     #ModoAutomatico;
      JU    END;
NETWORK
TITLE = END CASE
END:  NOP   0;
NETWORK
TITLE = Usita Digitale PlcOk
      AN    #AllarmeEmergenza;
      =     #DO_PlcOk;
END_FUNCTION

FUNCTION FC 21 : VOID
VERSION : 0.1
VAR_INPUT
  NumDBallarmi : BLOCK_DB ;
  Reset_Allarmi : BOOL ;
END_VAR
VAR_OUTPUT
  AllarmeEmergenza : BOOL ;
  AllarmeStopCiclo : BOOL ;
  AllarmeStartCiclo : BOOL ;
  AllarmeWarning : BOOL ;
END_VAR
VAR_TEMP
  Appoggio : ARRAY  [1 .. 8 ] OF BOOL ;
  Index : INT ;
END_VAR
BEGIN
NETWORK
TITLE = Allarmi Emergenza: Byte 0:7
      OPN   #NumDBallarmi;
      L     DBD 0;
      L     0;
      ==D;
      =     #Appoggio[1];
      L     DBD 4;
      L     0;
      ==D;
      =     #Appoggio[2];
      A     #Appoggio[1];
      A     #Appoggio[2];
      NOT;
      =     #AllarmeEmergenza;
NETWORK
TITLE = Allarmi StopCiclo: Byte 8:15
      L     DBD 8;
      L     0;
      ==D;
      =     #Appoggio[3];
      L     DBD 12;
      L     0;
      ==D;
      =     #Appoggio[4];
      A     #Appoggio[3];
      A     #Appoggio[4];
      NOT;
      O     #AllarmeEmergenza;
      =     #AllarmeStopCiclo;
NETWORK
TITLE = Allarmi StarCiclo: Byte 16:23
      L     DBD 16;
      L     0;
      ==D;
      =     #Appoggio[5];
      L     DBD 20;
      L     0;
      ==D;
      =     #Appoggio[6];
      A     #Appoggio[5];
      A     #Appoggio[6];
      NOT;
      O     #AllarmeEmergenza;
      =     #AllarmeStartCiclo;
NETWORK
TITLE = Allarmi Warning: Byte 24:30
      L     DBD 24;
      L     0;
      ==D;
      =     #Appoggio[7];
      L     DBD 28;
      L     0;
      ==D;
      =     #Appoggio[8];
      A     #Appoggio[7];
      A     #Appoggio[8];
      NOT;
      =     #AllarmeWarning;
NETWORK
TITLE = Reset di tutti gli Allarmi
      A     #Reset_Allarmi;
      JCN   end;
      L     8;
Znxt: T     #Index;
      L     1;
      -D;
      SLD   5;	//Colcolo l'indirizzo della DBD (#Index * 8 * 4)
      LAR1;
      L     0;
      T     DBD [AR1,P#0.0];
      L     #Index;
      LOOP  Znxt;
end:  NOP   0;
END_FUNCTION

// FC 40: know-how protected block, not included

FUNCTION FC 50 : VOID
VERSION : 0.1
VAR_TEMP
  Alarm_Emergency : BOOL ;
  Rich_manuale : BOOL ;
  Rich_automatico : BOOL ;
END_VAR
BEGIN
NETWORK
TITLE =
      CALL  FC 51;
      CALL  FC 53;
NETWORK
TITLE =
      CALL  FC 21 (
           NumDBallarmi             := DB 54,
           Reset_Allarmi            := DB55.DBX 0.0,
           AllarmeEmergenza         := DB50.DBX 2.0,
           AllarmeStopCiclo         := DB50.DBX 2.1,
           AllarmeStartCiclo        := DB50.DBX 2.2,
           AllarmeWarning           := DB50.DBX 2.3);
// cumula gli stati di emergenza per evitare definizioni errate degli stati macchina!
      A     DB50.DBX 2.0;
      O     DB100.DBX 2.0;
      O     DB150.DBX 2.0;
      O     DB200.DBX 2.0;
      =     #Alarm_Emergency;
      A     DB51.DBX 1.6;
      =     #Rich_manuale;
      A     DB51.DBX 1.7;
      A     DB55.DBX 10.1;
      =     #Rich_automatico;
      CALL  FC 20 (
           Enable                   := TRUE,
           AllarmeEmergenza         := #Alarm_Emergency,
           AusiliariOK              := DB51.DBX 0.4,
           ComandoTestMacchina      := FALSE,
           ComandoSetup             := FALSE,
           ComandoManuale           := #Rich_manuale,
           ComandoAutomatico        := #Rich_automatico,
           TimerTest                := T 1,
           ModoEmergenza            := DB50.DBX 0.0,
           ModoTestMacchina         := DB50.DBX 0.1,
           ModoSetup                := DB50.DBX 0.2,
           ModoManuale              := DB50.DBX 0.3,
           ModoAutomatico           := DB50.DBX 0.4,
           DO_PlcOk                 := DB55.DBX 10.0);
NETWORK
TITLE =
      CALL  FC 55;
      CALL  FC 70;
      CALL  FC 60;
NETWORK
TITLE =
      CALL  FC 52;
END_FUNCTION

FUNCTION FC 51 : VOID
VERSION : 0.1
BEGIN
NETWORK
TITLE =
      A     I 0.0;
      =     DB51.DBX 0.0;
      A     I 0.1;
      =     DB51.DBX 0.1;
      A     I 0.2;
      =     DB51.DBX 0.2;
      A     I 0.3;
      =     DB51.DBX 0.3;
      A     I 0.4;
      =     DB51.DBX 0.4;
      A     I 0.5;
      =     DB51.DBX 0.5;
      A     I 0.6;
      =     DB51.DBX 0.6;
      A     I 0.7;
      =     DB51.DBX 0.7;
NETWORK
TITLE =
      A     I 1.0;
      =     DB51.DBX 1.0;
      A     I 1.1;
      =     DB51.DBX 1.1;
      A     I 1.2;
      =     DB51.DBX 1.2;
      A     I 1.3;
      =     DB51.DBX 1.3;
      A     I 1.4;
      =     DB51.DBX 1.4;
      AN    I 1.5;
      =     DB51.DBX 1.5;
      A     I 1.7;
      =     DB51.DBX 1.6;
      A     I 1.6;
      =     DB51.DBX 1.7;
NETWORK
TITLE =
      A     I 2.0;
      =     DB51.DBX 2.0;
      A     I 2.1;
      =     DB51.DBX 2.1;
      A     I 6.2;
      =     DB51.DBX 2.2;
      A     I 6.3;
      =     DB51.DBX 2.3;
      A     I 6.4;
      =     DB51.DBX 2.4;
      A     I 6.5;
      =     DB51.DBX 2.5;
      A     I 7.6;
      =     DB51.DBX 2.6;
      A     I 7.5;
      =     DB51.DBX 2.7;
NETWORK
TITLE =
      A     I 6.6;
      =     DB51.DBX 3.0;
      A     I 2.2;
      =     DB51.DBX 3.1;
      A     I 4.7;
      =     DB51.DBX 3.2;
END_FUNCTION

FUNCTION FC 52 : VOID
VERSION : 0.1
BEGIN
NETWORK
TITLE =
      A     DB52.DBX 0.0;
      =     Q 0.0;
// tolto!
//      UN    "Line.MapA".Valvola_generale_aria
//      =     A      3.5
      A     DB52.DBX 0.2;
      =     Q 1.0;
      A     DB52.DBX 0.3;
      =     Q 1.1;
//      U     "Line.MapA".Spare_0_4
//      =     A      1.2
      A     DB52.DBX 0.5;
      =     Q 3.6;
      A     DB52.DBX 0.6;
      =     Q 3.7;
      A     DB52.DBX 0.7;
      =     Q 0.7;
      A     DB52.DBX 1.0;
      =     Q 1.7;
END_FUNCTION

FUNCTION FC 53 : VOID
VERSION : 0.1
BEGIN
NETWORK
TITLE =
      L     L#100;
      T     DB53.DBD 8;
      T     DB53.DBD 12;
// Impostate da pagina Config su OP
//      L     L#15000
//      T     "Line.Config".Vel_max_assi_auto
////      T     "Line.Config".Vel_max_assi_man
//      L     L#71501
//      T     "Line.Config".Offset_attrezzo_OP10_X
//      L     L#47116
//      T     "Line.Config".Offset_attrezzo_OP10_Y
//      L     L#371523
//      T     "Line.Config".Offset_attrezzo_OP40_X
//      L     L#47047
//      T     "Line.Config".Offset_attrezzo_OP40_Y
END_FUNCTION

FUNCTION FC 55 : VOID
VERSION : 0.1
VAR_TEMP
  Cmd_Marcia_ribaditrice : BOOL ;
  Cmd_Marcia_ribaditr_ibl : BOOL ;
  Cmd_abbassa_rib : BOOL ;
  Cmd_alza_rib : BOOL ;
  Cmd_abbassa_rib_ibl : BOOL ;
  Cmd_alza_rib_ibl : BOOL ;
  StartPosizX : BOOL ;
  StartPosizX_ibl : BOOL ;
  JogPiuX : BOOL ;
  JogMenoX : BOOL ;
  JogPiuX_ibl : BOOL ;
  JogMenoX_ibl : BOOL ;
  StartPosizY : BOOL ;
  StartPosizY_ibl : BOOL ;
  JogPiuY : BOOL ;
  JogMenoY : BOOL ;
  JogPiuY_ibl : BOOL ;
  JogMenoY_ibl : BOOL ;
  Profi_w_error : BOOL ;
  Profi_r_error : BOOL ;
  Override : INT ;
  Velocita_asse_X : DINT ;
  Velocita_asse_Y : DINT ;
  TeachIn_page_OP10 : BOOL ;
  TeachIn_page_OP40 : BOOL ;
  Punt1 : DINT ;
  PuntoSelezionato : INT ;
  Pos_comandata_asse_X : DINT ;
  Pos_comandata_asse_Y : DINT ;
  Tempo_ribaditura : DINT ;
END_VAR
BEGIN
NETWORK
TITLE = ******************       Diagnostica       *******************
NETWORK
TITLE = Diagnostica: Reset Allarmi
      A     DB51.DBX 2.4;
      FP    M 50.0;
      O(;
      A     DB70.DBX 16.0;
      FP    M 50.1;
      );
      S     DB55.DBX 0.0;
      A     DB55.DBX 0.0;
      L     S5T#500MS;
      SD    T 2;
      A     T 2;
      R     DB55.DBX 0.0;
NETWORK
TITLE = Allarmi di emergenza
      AN    DB51.DBX 0.1;
      O(;
      A     DB54.DBX 0.0;
      AN    DB55.DBX 0.0;
      );
      =     DB54.DBX 0.0;
      AN    DB51.DBX 0.2;
      O(;
      A     DB54.DBX 0.1;
      AN    DB55.DBX 0.0;
      );
      =     DB54.DBX 0.1;
      AN    DB51.DBX 0.7;
      O(;
      A     DB54.DBX 0.2;
      AN    DB55.DBX 0.0;
      );
      =     DB54.DBX 0.2;
      AN    DB51.DBX 2.0;
      O(;
      A     DB54.DBX 0.3;
      AN    DB55.DBX 0.0;
      );
      =     DB54.DBX 0.3;
      AN    DB51.DBX 2.1;
      O(;
      A     DB54.DBX 0.4;
      AN    DB55.DBX 0.0;
      );
      =     DB54.DBX 0.4;
      A     DB52.DBX 0.0;
      AN    DB51.DBX 1.0;
      O(;
      AN    DB52.DBX 0.0;
      A     DB51.DBX 1.0;
      );
      L     S5T#500MS;
      SD    T 3;
      A     T 3;
      S     DB54.DBX 1.5;
NETWORK
TITLE = Extracorsa Assi: Allarmi Emergenza
NETWORK
TITLE = Allarmi di STOP CICLO
      AN    DB51.DBX 0.4;
      =     DB54.DBX 9.2;
NETWORK
TITLE = Allarmi di NON START CICLO
NETWORK
TITLE = Allarmi di Warning
      AN    DB51.DBX 0.0;
//      O(    
//      U     DB54.DBX   24.0
//      UN    DB55.DBX    0.0
//      )     
      =     DB54.DBX 24.0;
      AN    DB51.DBX 0.3;
      =     DB54.DBX 24.1;
      A     DB51.DBX 0.6;
      =     DB54.DBX 24.2;
NETWORK
TITLE = Diagnostica: Hold Macchina
      AN    DB50.DBX 2.0;
      A(;
      A     DB50.DBX 0.4;
      AN    DB50.DBX 2.1;
      A     DB55.DBX 10.5;
      O(;
      A     DB50.DBX 0.3;
      A     DB55.DBX 10.1;
      );
      );
      =     DB50.DBX 2.4;
NETWORK
TITLE = ******************          Stati            *******************
      A     DB105.DBX 10.3;
      O     DB105.DBX 10.2;
      A     DB105.DBX 10.5;
      =     DB55.DBX 10.6;
      A     DB205.DBX 10.3;
      O     DB205.DBX 10.2;
      A     DB205.DBX 10.5;
      =     DB55.DBX 10.7;
NETWORK
TITLE =
      A     DB51.DBX 0.5;
      =     DB55.DBX 10.1;
NETWORK
TITLE = Stato: Fronte Start Ciclo
NETWORK
TITLE = Lampade
      AN    DB55.DBX 10.1;
      A     M 250.4;
      O     DB55.DBX 10.1;
      =     DB52.DBX 1.0;
NETWORK
TITLE = Pagina attiva di TeachIn
// Trovo quale stazione è in pagina di gestione punti
      L     DB70.DBW 0;
      L     21;
      ==I;
      =     #TeachIn_page_OP10;
      L     DB70.DBW 0;
      L     31;
      ==I;
      =     #TeachIn_page_OP40;
NETWORK
TITLE = ******************         Sistemi           *******************
NETWORK
TITLE = Uscita PLC OK
      A     DB55.DBX 10.0;
      =     DB52.DBX 0.0;
NETWORK
TITLE = Valvola generale aria
//      UN    "Line".Mode.Emergency
//      =     "Line.MapA".Valvola_generale_aria
      A     DB51.DBX 0.4;
      AN    DB51.DBX 3.0;
      O(;
      AN    DB51.DBX 0.4;
      A     DB51.DBX 3.0;
      );
      L     S5T#3S;
      SD    T 5;
      A     T 5;
      A     DB51.DBX 0.4;
      ON    DB51.DBX 2.5;
      O(;
      A     DB54.DBX 0.5;
      AN    DB55.DBX 0.0;
      );
      =     DB54.DBX 0.5;
      A     T 5;
      AN    DB51.DBX 0.4;
      O(;
      A     DB54.DBX 0.6;
      AN    DB55.DBX 0.0;
      );
      =     DB54.DBX 0.6;
NETWORK
TITLE = Prenotazione ribaditrice
      A     DB105.DBX 0.7;
      =     DB55.DBX 3.0;
      A     DB205.DBX 0.7;
      =     DB55.DBX 3.1;
      A     DB60.DBX 9.2;
      =     DB55.DBX 13.0;
      A     DB60.DBX 10.4;
      =     DB55.DBX 13.1;
NETWORK
TITLE = Marcia ribaditrice
//*************************** COMANDI DA CICLI *************************
      A     DB105.DBX 1.1;
      A     DB55.DBX 3.0;
      O(;
      A     DB205.DBX 1.1;
      A     DB55.DBX 3.1;
      );
      =     DB55.DBX 0.4;
//*************************** COMANDI SENZA INTERBLOCCHI ***************
// Autoritenuta comando di marcia manuale
      A     DB70.DBX 12.1;
      A     DB51.DBX 2.2;
      O     DB55.DBX 10.2;
      A     DB50.DBX 0.3;
      A(;
      AN    DB51.DBX 2.3;
      ON    DB70.DBX 12.1;
      );
      AN    DB54.DBX 24.4;
      A(;
      L     DB70.DBW 0;
      L     20;
      ==I;
      O(;
      L     DB70.DBW 0;
      L     30;
      ==I;
      );
      );
      =     DB55.DBX 0.5;
//CMD---------->Comando Marcia ribaditrice
//MANUALE
      A     DB55.DBX 0.5;
      A     DB50.DBX 0.3;
//AUTOMATICO
      O(;
      A     DB50.DBX 0.4;
      AN    DB50.DBX 2.6;
      A     DB55.DBX 0.4;
      );
//SICUREZZA
      A     DB50.DBX 2.4;
      A     DB51.DBX 0.0;
      =     #Cmd_Marcia_ribaditrice;
//************************** INTERBLOCCHI (E SEGNALAZIONE) ****************************
//MSG---> Segnalazione interblocco Movimento ribaditrice non ammesso con motore ribaditrice in marcia
//      U     "Line.Systems".Command.Reset_allarmi
//      O(    
//      U     "Line.Systems".State.Cassetto_OP10_indexato
//      U     "Line.Systems".State.Cassetto_OP40_indexato
//      )     
//      R     "Line.Alarms".Warning.Alarm05
//      U     #Cmd_Marcia_ribaditrice
//      U(    
//      UN    "Line.Systems".State.Cassetto_OP10_indexato
//      ON    "Line.Systems".State.Cassetto_OP40_indexato
//      )     
//      S     "Line.Alarms".Warning.Alarm05
//************************** COMANDI CON INTERBLOCCHI ******************************
//CMD-------------> Comando Marcia
      A     #Cmd_Marcia_ribaditrice;
      AN    DB54.DBX 24.4;
      =     #Cmd_Marcia_ribaditr_ibl;
      =     DB55.DBX 10.2;
      =     DB52.DBX 0.2;
NETWORK
TITLE = Alza/abbassa ribaditrice
//*************************** COMANDI DA CICLI *************************
      A     DB105.DBX 1.2;
      A     DB55.DBX 3.0;
      O(;
      A     DB205.DBX 1.2;
      A     DB55.DBX 3.1;
      );
      =     DB55.DBX 0.2;
      A     DB105.DBX 1.3;
      A     DB55.DBX 3.0;
      O(;
      A     DB205.DBX 1.3;
      A     DB55.DBX 3.1;
      );
      =     DB55.DBX 0.3;
//*************************** COMANDI SENZA INTERBLOCCHI ***************
//CMD---------->Comando abbassa ribaditrice
//MANUALE
      A     DB70.DBX 12.0;
      A     DB51.DBX 2.2;
      A     DB50.DBX 0.3;
//AUTOMATICO
      O(;
      A     DB50.DBX 0.4;
      AN    DB50.DBX 2.6;
      A     DB55.DBX 0.2;
      );
//SICUREZZA
      A     DB50.DBX 2.4;
      =     #Cmd_abbassa_rib;
//CMD---------->Comando alza ribaditrice
//MANUALE
      A     DB70.DBX 12.0;
      A     DB51.DBX 2.3;
      A     DB50.DBX 0.3;
//AUTOMATICO
      O(;
      A     DB50.DBX 0.4;
      AN    DB50.DBX 2.6;
      A     DB55.DBX 0.3;
      );
//SICUREZZA
      A     DB50.DBX 2.4;
      =     #Cmd_alza_rib;
//************************** INTERBLOCCHI (E SEGNALAZIONE) ****************************
//MSG---> Segnalazione interblocco Movimento ribaditrice non ammesso con motore ribaditrice in marcia
//      U     "Line.Systems".Command.Reset_allarmi
//      O     "Line.Systems".State.Ribadit_Motore_in_marcia
//      R     "Line.Alarms".Warning.Alarm04
//      U     #Cmd_abbassa_rib
//      O     #Cmd_alza_rib
//      Un    "Line.Systems".State.Ribadit_Motore_in_marcia
//      S     "Line.Alarms".Warning.Alarm04
      A     DB55.DBX 0.0;
      O(;
      A     DB55.DBX 10.6;
      A     DB55.DBX 10.7;
      );
      R     DB54.DBX 24.5;
      A     #Cmd_abbassa_rib;
      A(;
      AN    DB55.DBX 10.6;
      ON    DB55.DBX 10.7;
      );
      S     DB54.DBX 24.5;
//************************** COMANDI CON INTERBLOCCHI ******************************
//CMD-------------> Comando Mensola Contropunta SX
      AN    DB54.DBX 24.3;
      AN    DB54.DBX 24.5;
      A     #Cmd_abbassa_rib;
      =     #Cmd_abbassa_rib_ibl;
      AN    DB54.DBX 24.3;
      A     #Cmd_alza_rib;
      =     #Cmd_alza_rib_ibl;
      CALL  FB 102 , DB 400 (
           DIX 0.0                  := TRUE,
           DIX 0.1                  := #Cmd_abbassa_rib_ibl,
           DIX 0.2                  := #Cmd_alza_rib_ibl,
           DIX 0.3                  := DB51.DBX 2.6,
           DIX 0.4                  := DB51.DBX 2.7,
           DIX 0.5                  := DB55.DBX 0.0,
           DID 2                    := L#4000,
           DIX 6.0                  := FALSE,
           DIX 8.0                  := DB52.DBX 0.3,
           DIX 8.2                  := DB55.DBX 10.3,
           DIX 8.3                  := DB55.DBX 10.4,
           DIX 8.4                  := DB54.DBX 8.0,
           DIX 8.5                  := DB54.DBX 8.1,
           DIX 8.6                  := DB54.DBX 8.2);
NETWORK
TITLE = Blocco porte
//************************************* COMANDI ***************************************
      A     DB50.DBX 0.4;
      A     DB55.DBX 10.1;
      =     DB52.DBX 0.5;
      =     DB52.DBX 0.6;
//************************** INTERBLOCCHI (E SEGNALAZIONE) ****************************
// Allamre porte non chiuse
      A     DB55.DBX 0.0;
      O     DB50.DBX 0.3;
      R     DB54.DBX 8.3;
      A     DB50.DBX 0.4;
      AN    DB55.DBX 10.1;
      S     DB54.DBX 8.3;
// Allarme porte non bloccate
      A     DB55.DBX 0.0;
      O     DB50.DBX 0.3;
      R     DB54.DBX 8.4;
      R     DB54.DBX 8.5;
      A     DB52.DBX 0.5;
      O     DB52.DBX 0.6;
      L     S5T#1S;
      SD    T 6;
      A     T 6;
      AN    DB51.DBX 1.1;
      S     DB54.DBX 8.4;
      A     T 6;
      AN    DB51.DBX 1.2;
      S     DB54.DBX 8.5;
//************************************* STATI ***************************************
      A     DB52.DBX 0.5;
      A     DB52.DBX 0.6;
      AN    DB54.DBX 8.3;
      AN    DB54.DBX 8.4;
      AN    DB54.DBX 8.5;
      =     DB55.DBX 10.5;
NETWORK
TITLE = Input asse X
      CALL  FB 455 , DB 425 (
           DIX 0.0                  := TRUE,
           DIW 2                    := 400,
           DIW 4                    := 400,
           DIX 6.1                  := DB55.DBX 11.4,
           DIX 8.0                  := #Profi_w_error,
           DIX 8.1                  := #Profi_r_error);	// indirizzo 400
      A     #Profi_w_error;
      O     #Profi_r_error;
      S     DB54.DBX 1.1;
      AN    DB55.DBX 11.4;
      O     DB51.DBX 3.1;
      AN    #Profi_w_error;
      AN    #Profi_r_error;
      S     DB54.DBX 1.3;
NETWORK
TITLE = Input asse Y
      CALL  FB 455 , DB 426 (
           DIX 0.0                  := TRUE,
           DIW 2                    := 430,
           DIW 4                    := 430,
           DIX 6.1                  := DB55.DBX 12.4,
           DIX 8.0                  := #Profi_w_error,
           DIX 8.1                  := #Profi_r_error);	// indirizzo 430
      A     #Profi_w_error;
      O     #Profi_r_error;
      S     DB54.DBX 1.2;
      AN    DB55.DBX 12.4;
      O     DB51.DBX 3.2;
      AN    #Profi_w_error;
      AN    #Profi_r_error;
      S     DB54.DBX 1.4;
NETWORK
TITLE = Asse X
//*************************** COMANDI DA CICLI *************************
      AN    DB55.DBX 0.0;
      O     DB55.DBX 11.7;
      A     DB50.DBX 2.4;
      A     DB55.DBX 11.4;
      AN    DB51.DBX 3.1;
      =     DB55.DBX 1.0;
      A     DB105.DBX 1.0;
      A     DB55.DBX 13.0;
      O(;
      A     DB205.DBX 1.0;
      A     DB55.DBX 13.1;
      );
      A     DB55.DBX 11.4;
      A     DB55.DBX 1.0;
      A     DB55.DBX 11.7;
      =     DB55.DBX 1.1;
//*************************** COMANDI SENZA INTERBLOCCHI ***************
//CMD---------->Comando posiziona
//MANUALE
      A     #TeachIn_page_OP10;
      O     #TeachIn_page_OP40;
      A     DB70.DBX 16.1;
      A     DB50.DBX 0.3;
//AUTOMATICO
      O(;
      A     DB50.DBX 0.4;
      AN    DB50.DBX 2.6;
      A     DB55.DBX 1.1;
      );
//SICUREZZA
      A     DB50.DBX 2.4;
      =     #StartPosizX;
//CMD---------->Comando Jog +
//MANUALE
      A     DB70.DBX 12.2;
      A     DB51.DBX 2.2;
      A     DB50.DBX 0.3;
//AUTOMATICO
//SICUREZZA
      A     DB50.DBX 2.4;
      =     #JogPiuX;
//CMD---------->Comando Jog -
//MANUALE
      A     DB70.DBX 12.2;
      A     DB51.DBX 2.3;
      A     DB50.DBX 0.3;
//AUTOMATICO
//SICUREZZA
      A     DB50.DBX 2.4;
      =     #JogMenoX;
//************************** INTERBLOCCHI (E SEGNALAZIONE) ****************************
//MSG---> Segnalazione interblocco
      A     DB55.DBX 0.0;
      O     DB55.DBX 10.4;
      R     DB54.DBX 8.6;
      A     #StartPosizX;
      O     #JogPiuX;
      O     #JogMenoX;
      AN    DB55.DBX 10.4;
      S     DB54.DBX 8.6;
      A     DB55.DBX 0.0;
      O(;
      A     DB55.DBX 10.6;
      A     DB55.DBX 10.7;
      );
      R     DB54.DBX 24.6;
      A     #StartPosizX;
      O     #JogPiuX;
      O     #JogMenoX;
      A(;
      AN    DB55.DBX 10.6;
      ON    DB55.DBX 10.7;
      );
      S     DB54.DBX 24.6;
//************************** COMANDI CON INTERBLOCCHI ******************************
      AN    DB54.DBX 8.6;
      AN    DB54.DBX 24.6;
      A     #StartPosizX;
      =     #StartPosizX_ibl;
      AN    DB54.DBX 8.6;
      AN    DB54.DBX 24.6;
      A     #JogPiuX;
      =     #JogPiuX_ibl;
      AN    DB54.DBX 8.6;
      AN    DB54.DBX 24.6;
      A     #JogMenoX;
      =     #JogMenoX_ibl;
//*********************************  OVERRIDE  *************************************
      L     DB70.DBW 48;
      A     DB50.DBX 0.3;
      JC    Ovx;
      L     DB70.DBW 50;
      A     DB50.DBX 0.4;
      JC    Ovx;
      L     0;
Ovx:  T     #Override;
//*********************************  POSIZIONE  *************************************
      A     DB55.DBX 13.0;
      A     DB105.DBX 1.0;
      A     DB50.DBX 0.4;
      JCN   nX10;
      L     DB105.DBD 22;
      L     DB53.DBD 16;
      +D;
      T     DB55.DBD 30;
      JU    EnX;
nX10: A     DB55.DBX 13.1;
      A     DB205.DBX 1.0;
      A     DB50.DBX 0.4;
      JCN   nX40;
      L     DB205.DBD 22;
      L     DB53.DBD 24;
      +D;
      T     DB55.DBD 30;
      JU    EnX;
nX40: A     #TeachIn_page_OP10;
      A     DB70.DBX 16.1;
      A     DB50.DBX 0.3;
      JCN   nXv1;
      L     DB70.DBD 74;
      L     DB53.DBD 16;
      +D;
      T     DB55.DBD 30;
      JU    EnX;
nXv1: A     #TeachIn_page_OP40;
      A     DB70.DBX 16.1;
      A     DB50.DBX 0.3;
      JCN   nXv4;
      L     DB70.DBD 74;
      L     DB53.DBD 24;
      +D;
      T     DB55.DBD 30;
      JU    EnX;
nXv4: NOP   0;
// Errore di comando posizione
      L     0;
      T     DB55.DBD 30;
EnX:  NOP   0;
//*********************************  VELOCITA'  *************************************
// limita velocità massima di ricetta
      A     DB55.DBX 13.1;
      JC    x40;
      L     DB110.DBD 40;
      T     #Velocita_asse_X;
      JU    x10;
x40:  L     DB210.DBD 40;
      T     #Velocita_asse_X;
x10:  NOP   0;
      L     #Velocita_asse_X;
      L     DB53.DBD 0;
      <D;
      JC    m1x;
      L     DB53.DBD 0;
      T     #Velocita_asse_X;
m1x:  NOP   0;
// imposta velcità automatico
      A     DB50.DBX 0.4;
      JCN   nVaX;
      L     #Velocita_asse_X;
      T     DB55.DBD 26;
      L     DB53.DBD 8;
      T     DB55.DBW 22;
      T     DB55.DBW 24;
      JU    nVmX;
// imposta velocità manuale
nVaX: L     DB53.DBD 4;
      T     DB55.DBD 26;
      L     DB53.DBD 12;
      T     DB55.DBW 22;
      T     DB55.DBW 24;
nVmX: NOP   0;
      CALL  FB 450 , DB 420 (
           DIX 0.0                  := TRUE,
           DIW 2                    := 404,
           DIW 4                    := 404,
           DIX 6.0                  := #JogMenoX_ibl,
           DIX 6.1                  := #JogPiuX_ibl,
           DIX 6.2                  := #StartPosizX_ibl,
           DIX 6.3                  := M 10.0,
           DIX 6.4                  := M 10.1,
           DIX 6.5                  := DB55.DBX 1.0,
           DIX 6.6                  := DB55.DBX 0.0,
           DIW 8                    := #Override,
           DIW 10                   := DB55.DBW 22,
           DIW 12                   := DB55.DBW 24,
           DID 14                   := DB55.DBD 26,
           DID 18                   := DB55.DBD 30,
           DIW 22                   := 0,
           DIX 24.0                 := #Profi_w_error,
           DIX 24.1                 := #Profi_r_error,
           DIX 24.2                 := DB55.DBX 11.0,
           DIX 24.3                 := DB55.DBX 11.1,
           DIX 24.4                 := DB55.DBX 11.2,
           DIB 25                   := DB55.DBB 38,
           DID 26                   := DB55.DBD 34,
           DIX 30.0                 := DB55.DBX 11.6,
           DIX 30.1                 := DB55.DBX 11.5,
           DIX 30.2                 := DB55.DBX 11.7);	// indirizzo 404
      A     #Profi_w_error;
      O     #Profi_r_error;
      S     DB54.DBX 0.7;
NETWORK
TITLE = Asse Y
//*************************** COMANDI DA CICLI *************************
      AN    DB55.DBX 0.0;
      O     DB55.DBX 12.7;
      A     DB50.DBX 2.4;
      A     DB55.DBX 12.4;
      AN    DB51.DBX 3.2;
      =     DB55.DBX 2.0;
      A     DB105.DBX 1.0;
      A     DB55.DBX 13.0;
      O(;
      A     DB205.DBX 1.0;
      A     DB55.DBX 13.1;
      );
      A     DB55.DBX 12.4;
      A     DB55.DBX 2.0;
      A     DB55.DBX 12.7;
      =     DB55.DBX 2.1;
//*************************** COMANDI SENZA INTERBLOCCHI ***************
//CMD---------->Comando posiziona
//MANUALE
      A     #TeachIn_page_OP10;
      O     #TeachIn_page_OP40;
      A     DB70.DBX 16.1;
      A     DB50.DBX 0.3;
//AUTOMATICO
      O(;
      A     DB50.DBX 0.4;
      AN    DB50.DBX 2.6;
      A     DB55.DBX 2.1;
      );
//SICUREZZA
      A     DB50.DBX 2.4;
      =     #StartPosizY;
//CMD---------->Comando Jog +
//MANUALE
      A     DB70.DBX 12.3;
      A     DB51.DBX 2.2;
      A     DB50.DBX 0.3;
//AUTOMATICO
//SICUREZZA
      A     DB50.DBX 2.4;
      =     #JogPiuY;
//CMD---------->Comando Jog -
//MANUALE
      A     DB70.DBX 12.3;
      A     DB51.DBX 2.3;
      A     DB50.DBX 0.3;
//AUTOMATICO
//SICUREZZA
      A     DB50.DBX 2.4;
      =     #JogMenoY;
//************************** INTERBLOCCHI (E SEGNALAZIONE) ****************************
//MSG---> Segnalazione interblocco
      A     DB55.DBX 0.0;
      O     DB55.DBX 10.4;
      R     DB54.DBX 8.7;
      A     #StartPosizY;
      O     #JogPiuY;
      O     #JogMenoY;
      AN    DB55.DBX 10.4;
      S     DB54.DBX 8.7;
// una segnalazione per entrambi gli assi: reset su gestione asse X
      A     #StartPosizY;
      O     #JogPiuY;
      O     #JogMenoY;
      A(;
      AN    DB55.DBX 10.6;
      ON    DB55.DBX 10.7;
      );
      S     DB54.DBX 24.6;
//************************** COMANDI CON INTERBLOCCHI ******************************
      AN    DB54.DBX 8.7;
      AN    DB54.DBX 24.6;
      A     #StartPosizY;
      =     #StartPosizY_ibl;
      AN    DB54.DBX 8.7;
      AN    DB54.DBX 24.6;
      A     #JogPiuY;
      =     #JogPiuY_ibl;
      AN    DB54.DBX 8.7;
      AN    DB54.DBX 24.6;
      A     #JogMenoY;
      =     #JogMenoY_ibl;
//*********************************  OVERRIDE  *************************************
      L     DB70.DBW 48;
      A     DB50.DBX 0.3;
      JC    Ovy;
      L     DB70.DBW 50;
      A     DB50.DBX 0.4;
      JC    Ovy;
      L     0;
Ovy:  T     #Override;
//*********************************  POSIZIONE  *************************************
      A     DB55.DBX 13.0;
      A     DB105.DBX 1.0;
      A     DB50.DBX 0.4;
      JCN   nY10;
      L     DB105.DBD 26;
      L     DB53.DBD 20;
      +D;
      T     DB55.DBD 60;
      JU    EnY;
nY10: A     DB55.DBX 13.1;
      A     DB205.DBX 1.0;
      A     DB50.DBX 0.4;
      JCN   nY40;
      L     DB205.DBD 26;
      L     DB53.DBD 28;
      +D;
      T     DB55.DBD 60;
      JU    EnY;
nY40: A     #TeachIn_page_OP10;
      A     DB70.DBX 16.1;
      A     DB50.DBX 0.3;
      JCN   nYv1;
      L     DB70.DBD 78;
      L     DB53.DBD 20;
      +D;
      T     DB55.DBD 60;
      JU    EnY;
nYv1: A     #TeachIn_page_OP40;
      A     DB70.DBX 16.1;
      A     DB50.DBX 0.3;
      JCN   nYv4;
      L     DB70.DBD 78;
      L     DB53.DBD 28;
      +D;
      T     DB55.DBD 60;
      JU    EnY;
nYv4: NOP   0;
// Errore di comando posizione
      L     0;
      T     DB55.DBD 60;
EnY:  NOP   0;
//*********************************  VELOCITA'  *************************************
// limita velocità massima di ricetta
      A     DB55.DBX 13.1;
      JC    y40;
      L     DB110.DBD 44;
      T     #Velocita_asse_Y;
      JU    y10;
y40:  L     DB210.DBD 44;
      T     #Velocita_asse_Y;
y10:  NOP   0;
      L     #Velocita_asse_Y;
      L     DB53.DBD 0;
      <D;
      JC    m1Y;
      L     DB53.DBD 0;
      T     #Velocita_asse_Y;
m1Y:  NOP   0;
// imposta velcità automatico
      A     DB50.DBX 0.4;
      JCN   nVaY;
      L     #Velocita_asse_Y;
      T     DB55.DBD 56;
      L     DB53.DBD 8;
      T     DB55.DBW 52;
      T     DB55.DBW 54;
      JU    nVmY;
// imposta velocità manuale
nVaY: L     DB53.DBD 4;
      T     DB55.DBD 56;
      L     DB53.DBD 12;
      T     DB55.DBW 52;
      T     DB55.DBW 54;
nVmY: NOP   0;
      CALL  FB 450 , DB 421 (
           DIX 0.0                  := TRUE,
           DIW 2                    := 434,
           DIW 4                    := 434,
           DIX 6.0                  := #JogMenoY_ibl,
           DIX 6.1                  := #JogPiuY_ibl,
           DIX 6.2                  := #StartPosizY_ibl,
           DIX 6.3                  := M 10.2,
           DIX 6.4                  := M 10.3,
           DIX 6.5                  := DB55.DBX 2.0,
           DIX 6.6                  := DB55.DBX 0.0,
           DIW 8                    := #Override,
           DIW 10                   := DB55.DBW 52,
           DIW 12                   := DB55.DBW 54,
           DID 14                   := DB55.DBD 56,
           DID 18                   := DB55.DBD 60,
           DIW 22                   := 0,
           DIX 24.0                 := #Profi_w_error,
           DIX 24.1                 := #Profi_r_error,
           DIX 24.2                 := DB55.DBX 12.0,
           DIX 24.3                 := DB55.DBX 12.1,
           DIX 24.4                 := DB55.DBX 12.2,
           DIB 25                   := DB55.DBB 68,
           DID 26                   := DB55.DBD 64,
           DIX 30.0                 := DB55.DBX 12.6,
           DIX 30.1                 := DB55.DBX 12.5,
           DIX 30.2                 := DB55.DBX 12.7);	// indirizzo 434
      A     #Profi_w_error;
      O     #Profi_r_error;
      S     DB54.DBX 0.7;
NETWORK
TITLE = Gestioen bit "Vai al punto" da TeachIn page
      AN    DB55.DBX 12.2;
      AN    DB55.DBX 11.2;
      A     DB70.DBX 16.1;
      L     S5T#500MS;
      SD    T 15;
      AN    #TeachIn_page_OP10;
      AN    #TeachIn_page_OP40;
      O     T 15;
      O     DB51.DBX 1.5;
      R     DB70.DBX 16.1;
NETWORK
TITLE = Leggi punto TeachIn page
// catturo momento di ingresso in pagina di teachIn
      A     #TeachIn_page_OP10;
      O     #TeachIn_page_OP40;
      FP    M 51.2;
      =     DB55.DBX 13.2;
// Modificato numero del punto
      L     DB70.DBW 68;
      L     DB55.DBW 80;
      <>I;
      =     DB55.DBX 13.3;
      L     DB70.DBW 68;
      T     DB55.DBW 80;
// Richiesta lettura punto da operatore
      A     DB70.DBX 16.4;
      FP    M 51.3;
      =     DB55.DBX 13.4;
      A     DB70.DBX 16.4;
      R     DB70.DBX 16.4;
// Funzione di lettura dei dati del punto selezionato
      A     DB55.DBX 13.2;
      O     DB55.DBX 13.3;
      O     DB55.DBX 13.4;
      JCN   noLP;
// Azzero le variabili
      L     L#0;
      T     DB70.DBD 74;
      T     DB70.DBD 78;
      T     DB70.DBD 82;
// controllo di esser in tabella (punto coerente)
      L     DB70.DBW 68;
      L     DB70.DBW 70;
      <I;
      O(;
      L     DB70.DBW 68;
      L     DB70.DBW 72;
      >I;
      );
      JC    noLP;
// Sceglie tabella in funzione della stazione OP10 o OP40
      L     DB70.DBW 68;
      T     #PuntoSelezionato;
      A     #TeachIn_page_OP40;
      JC    op2;
      OPN   DB 110;
      JU    op1;
op2:  OPN   DB 210;
op1:  NOP   0;
// Leggo i dati del punto
      L     #PuntoSelezionato;
      L     1;
      -I;
      ITD;
      L     L#12;
      *D;
      L     L#82;
      +D;
      SLW   3;
      T     #Punt1;
      L     DBD [#Punt1];
      T     #Pos_comandata_asse_X;
      L     #Punt1;
      L     32;
      +D;
      T     #Punt1;
      L     DBD [#Punt1];
      T     #Pos_comandata_asse_Y;
      L     #Punt1;
      L     32;
      +D;
      T     #Punt1;
      L     DBD [#Punt1];
      T     #Tempo_ribaditura;
      L     #Pos_comandata_asse_X;
      T     DB70.DBD 74;
      L     #Pos_comandata_asse_Y;
      T     DB70.DBD 78;
      L     #Tempo_ribaditura;
      T     DB70.DBD 82;
noLP: NOP   0;
NETWORK
TITLE = teachIn punto
// Richiesta TeachIn punto da operatore
      A     DB70.DBX 16.2;
      FP    M 51.5;
      =     DB55.DBX 13.6;
      A     DB70.DBX 16.2;
      R     DB70.DBX 16.2;
// Funzione di TeachIn del punto selezionato
      A     DB55.DBX 13.6;
      JCN   noTI;
      AN    #TeachIn_page_OP10;
      JC    NT10;
//OP10
      L     DB70.DBD 52;
      T     DB70.DBD 74;
      L     DB70.DBD 56;
      T     DB70.DBD 78;
      JU    noTI;
NT10: AN    #TeachIn_page_OP40;
      JC    NT40;
//OP40
      L     DB70.DBD 60;
      T     DB70.DBD 74;
      L     DB70.DBD 64;
      T     DB70.DBD 78;
NT40: NOP   0;
noTI: NOP   0;
NETWORK
TITLE = Salva punto
// Richiesta scrittura punto da operatore
      A     DB70.DBX 16.3;
      FP    M 51.4;
      =     DB55.DBX 13.5;
      A     DB70.DBX 16.3;
      R     DB70.DBX 16.3;
// Funzione di lettura dei dati del punto selezionato
      A     DB55.DBX 13.5;
      JCN   noSP;
// controllo di esser in tabella (punto coerente)
      L     DB70.DBW 68;
      L     DB70.DBW 70;
      <I;
      O(;
      L     DB70.DBW 68;
      L     DB70.DBW 72;
      >I;
      );
      JC    noSP;
// Sceglie tabella in funzione della stazione OP10 o OP40
// Salvo i dati del punto
      L     DB70.DBD 74;
      T     #Pos_comandata_asse_X;
      L     DB70.DBD 78;
      T     #Pos_comandata_asse_Y;
      L     DB70.DBD 82;
      T     #Tempo_ribaditura;
      L     DB70.DBW 68;
      T     #PuntoSelezionato;
      A     #TeachIn_page_OP40;
      JC    opS2;
      OPN   DB 110;
      JU    opS1;
opS2: OPN   DB 210;
opS1: NOP   0;
      L     #PuntoSelezionato;
      L     1;
      -I;
      ITD;
      L     L#12;
      *D;
      L     L#82;
      +D;
      SLW   3;
      T     #Punt1;
      L     #Pos_comandata_asse_X;
      T     DBD [#Punt1];
      L     #Punt1;
      L     32;
      +D;
      T     #Punt1;
      L     #Pos_comandata_asse_Y;
      T     DBD [#Punt1];
      L     #Punt1;
      L     32;
      +D;
      T     #Punt1;
      L     #Tempo_ribaditura;
      T     DBD [#Punt1];
noSP: NOP   0;
END_FUNCTION

FUNCTION FC 60 : VOID
VERSION : 0.1
BEGIN
NETWORK
TITLE =
NETWORK
TITLE =
      A     DB50.DBX 0.4;
      AN    DB50.DBX 2.1;
      AN    DB50.DBX 2.0;
// condizione di sicurezza
      =     DB60.DBX 18.0;
      CLR;
      =     DB50.DBX 2.6;
      CALL  FB 60 , DB 440 (
           DIX 0.0                  := DB60.DBX 18.0,
           DIX 0.1                  := DB50.DBX 2.6,
           DIX 0.2                  := FALSE,
           DIX 2.0                  := DB60.DBX 6.0,
           DIX 2.1                  := DB60.DBX 6.1,
           DIX 2.2                  := DB60.DBX 6.2,
           DIW 4                    := DB60.DBW 0,
           DIW 6                    := DB60.DBW 2,
           DIW 8                    := DB60.DBW 4);
END_FUNCTION

FUNCTION FC 70 : VOID
VERSION : 0.1
VAR_TEMP
  PagManualeVis : BOOL ;
  PagAutomaticoVis : BOOL ;
END_VAR
BEGIN
NETWORK
TITLE = Controlla pagina attiva
// Contollo se visualizzata una pagina automatica o manuale
      L     DB70.DBW 0;
      L     90;
      <=I;
      =     #PagManualeVis;
      L     DB70.DBW 0;
      L     199;
      <=I;
      A(;
      L     DB70.DBW 0;
      L     110;
      >=I;
      );
      =     #PagAutomaticoVis;
NETWORK
TITLE = Forza pagina attva
// Forzo le pagine principali in funzione dello modo abilitato
      A     DB50.DBX 0.4;
      A     #PagManualeVis;
      JC    FAu;
      A     DB50.DBX 0.3;
      A     #PagAutomaticoVis;
      JC    FMa;
      JU    NoF;
FAu:  L     120;
      T     DB70.DBW 10;
      JU    NoF;
FMa:  L     10;
      T     DB70.DBW 10;
NoF:  NOP   0;
NETWORK
TITLE = Visualizzazione stati sensori
      A     DB55.DBX 10.4;
      =     DB70.DBX 26.0;
      A     DB55.DBX 10.3;
      =     DB70.DBX 26.1;
      AN    DB55.DBX 10.2;
      =     DB70.DBX 26.2;
      A     DB55.DBX 10.2;
      =     DB70.DBX 26.3;
      A     DB105.DBX 10.4;
      =     DB70.DBX 26.4;
      A     DB105.DBX 10.5;
      =     DB70.DBX 26.5;
      A     DB105.DBX 10.6;
      =     DB70.DBX 26.6;
      A     DB105.DBX 10.7;
      =     DB70.DBX 26.7;
      A     DB55.DBX 11.5;
      =     DB70.DBX 27.0;
      A     DB55.DBX 11.6;
      =     DB70.DBX 27.1;
      A     DB55.DBX 12.5;
      =     DB70.DBX 27.2;
      A     DB55.DBX 12.6;
      =     DB70.DBX 27.3;
      A     DB155.DBX 10.4;
      =     DB70.DBX 27.4;
      A     DB155.DBX 10.5;
      =     DB70.DBX 27.5;
      A     DB155.DBX 10.6;
      =     DB70.DBX 27.6;
      A     DB155.DBX 10.7;
      =     DB70.DBX 27.7;
      A     DB155.DBX 11.0;
      =     DB70.DBX 28.0;
      A     DB155.DBX 11.1;
      =     DB70.DBX 28.1;
      A     DB205.DBX 10.4;
      =     DB70.DBX 28.2;
      A     DB205.DBX 10.5;
      =     DB70.DBX 28.3;
      A     DB205.DBX 10.6;
      =     DB70.DBX 28.4;
      A     DB205.DBX 10.7;
      =     DB70.DBX 28.5;
NETWORK
TITLE = Visualizzazione variabili macchina
// Visualizzazione assi
      L     DB55.DBD 34;
      T     DB70.DBD 36;
      L     DB55.DBD 64;
      T     DB70.DBD 40;
// Visualizzazione assi su OP10
      L     DB55.DBD 34;
      L     DB53.DBD 16;
      -D;
      T     DB70.DBD 52;
      L     DB55.DBD 64;
      L     DB53.DBD 20;
      -D;
      T     DB70.DBD 56;
// Visualizzazione assi su OP40
      L     DB55.DBD 34;
      L     DB53.DBD 24;
      -D;
      T     DB70.DBD 60;
      L     DB55.DBD 64;
      L     DB53.DBD 28;
      -D;
      T     DB70.DBD 64;
// Visualizzazione posizione punzone di piantaggio
      L     DB151.DBD 6;
      T     DB70.DBD 44;
NETWORK
TITLE = Stato macchina
      L     0;
      A     DB50.DBX 0.0;
      JC    cls;
      L     1;
      A     DB50.DBX 0.1;
      JC    cls;
      L     2;
      A     DB50.DBX 0.2;
      JC    cls;
      L     3;
      A     DB50.DBX 0.3;
      JC    cls;
      L     4;
      A     DB50.DBX 0.4;
      JC    cls;
      L     0;
cls:  T     DB70.DBW 162;
NETWORK
TITLE = Stati cicli
      A     DB120.DBX 18.0;
      =     DB70.DBX 150.0;
      A     DB120.DBX 40.0;
      =     DB70.DBX 150.1;
      A     DB170.DBX 18.0;
      =     DB70.DBX 150.2;
      A     DB170.DBX 40.0;
      =     DB70.DBX 150.3;
      A     DB220.DBX 18.0;
      =     DB70.DBX 150.4;
      A     DB220.DBX 40.0;
      =     DB70.DBX 150.5;
      A     DB120.DBX 40.0;
      JC    R10;
      L     DB120.DBW 4;
      T     DB70.DBW 152;
      JU    M10;
R10:  L     DB120.DBW 26;
      T     DB70.DBW 152;
M10:  NOP   0;
      L     DB105.DBW 20;
      T     DB70.DBW 154;
      A     DB170.DBX 40.0;
      JC    R20;
      L     DB170.DBW 4;
      T     DB70.DBW 160;
      JU    M20;
R20:  L     DB170.DBW 26;
      T     DB70.DBW 160;
M20:  NOP   0;
      A     DB220.DBX 40.0;
      JC    R40;
      L     DB220.DBW 4;
      T     DB70.DBW 156;
      JU    M40;
R40:  L     DB220.DBW 26;
      T     DB70.DBW 156;
M40:  NOP   0;
      L     DB205.DBW 20;
      T     DB70.DBW 158;
NETWORK
TITLE = Min / Max punto in teachIn in funzione della ricetta
      L     DB70.DBW 0;
      L     21;
      <>I;
      JC    n10;
      L     1;
      T     DB70.DBW 70;
      L     DB110.DBW 80;
      T     DB70.DBW 72;
      JU    n0;
n10:  L     DB70.DBW 0;
      L     31;
      <>I;
      JC    n40;
      L     1;
      T     DB70.DBW 70;
      L     DB210.DBW 80;
      T     DB70.DBW 72;
      JU    n0;
n40:  L     1;
      T     DB70.DBW 70;
      T     DB70.DBW 72;
n0:   NOP   0;
END_FUNCTION

FUNCTION FC 100 : VOID
VERSION : 0.1
VAR_TEMP
  ErrorToolType : BOOL ;
END_VAR
BEGIN
NETWORK
TITLE =
NETWORK
TITLE =
      CALL  FC 101;
      CALL  FC 106 (
           ToolType                 := DB110.DBW 34,
           ErrorToolType            := #ErrorToolType);
      A     #ErrorToolType;
      AN    DB110.DBX 78.0;
//      S     DB104.DBX    0.0
      S     DB104.DBX 9.0;
      CALL  FC 103;
NETWORK
TITLE =
      A     DB55.DBX 0.0;
      =     DB105.DBX 0.0;
      A     DB55.DBX 0.1;
      =     DB105.DBX 0.1;
      A     DB55.DBX 10.1;
      =     DB105.DBX 10.0;
      A     DB55.DBX 10.5;
      =     DB105.DBX 10.1;
      CALL  FC 21 (
           NumDBallarmi             := DB 104,
           Reset_Allarmi            := DB105.DBX 0.0,
           AllarmeEmergenza         := DB100.DBX 2.0,
           AllarmeStopCiclo         := DB100.DBX 2.1,
           AllarmeStartCiclo        := DB100.DBX 2.2,
           AllarmeWarning           := DB100.DBX 2.3);
// Bench mode = Line mode...
      A     DB50.DBX 0.0;
      =     DB100.DBX 0.0;
      A     DB50.DBX 0.1;
      =     DB100.DBX 0.1;
      A     DB50.DBX 0.2;
      =     DB100.DBX 0.2;
      A     DB50.DBX 0.3;
      =     DB100.DBX 0.3;
      A     DB50.DBX 0.4;
      =     DB100.DBX 0.4;
NETWORK
TITLE =
      CALL  FC 105;
      CALL  FC 120;
//      CALL  "Op10.Operator_Panel"
NETWORK
TITLE =
      CALL  FC 102;
END_FUNCTION

FUNCTION FC 101 : VOID
VERSION : 0.1
BEGIN
NETWORK
TITLE =
      A     I 6.0;
      =     DB101.DBX 0.0;
      AN    I 8.0;
      =     DB101.DBX 0.1;
      A     I 8.1;
      =     DB101.DBX 0.2;
      A     I 8.3;
      =     DB101.DBX 0.3;
      A     I 8.2;
      =     DB101.DBX 0.4;
      A     I 8.5;
      =     DB101.DBX 0.5;
      A     I 8.4;
      =     DB101.DBX 0.6;
      AN    I 1.5;
      =     DB101.DBX 0.7;
END_FUNCTION

FUNCTION FC 102 : VOID
VERSION : 0.1
BEGIN
NETWORK
TITLE =
      A     DB102.DBX 0.0;
      =     Q 0.3;
      A     DB102.DBX 0.1;
      =     Q 0.4;
      A     DB102.DBX 0.2;
      =     Q 2.2;
      A     DB102.DBX 0.3;
      =     Q 2.3;
      A     DB102.DBX 0.4;
      =     Q 2.5;
      A     DB102.DBX 0.5;
      =     Q 2.4;
END_FUNCTION

FUNCTION FC 103 : VOID
VERSION : 0.1
BEGIN
NETWORK
TITLE =
END_FUNCTION

